// TIA Portal project "CommRS485" (V17)

(* hardware
DEVICE "S7-1200 station_1"  S7-1200 Station
   slot 0: "Rack_0"  S7-1200 Rack  Rack  V1.0
   slot 1: "PLC_1"  CPU 1211C DC/DC/Rly  6ES7 211-1HE40-0XB0  V4.5
   slot 101: "CM 1241 (RS422/485)_1"  6ES7 241-1CH32-0XB0  V2.2
DEVICE "S7-1200 station_2"  S7-1200 Station
   slot 0: "Rack_0"  S7-1200 Rack  Rack  V1.0
   slot 1: "PLC_2"  CPU 1211C DC/DC/Rly  6ES7 211-1HE40-0XB0  V4.5
   slot 101: "CM 1241 (RS422/485)_1"  6ES7 241-1CH32-0XB0  V2.2
DEVICE "S7-1200 station_3"  S7-1200 Station
   slot 0: "Rack_0"  S7-1200 Rack  Rack  V1.0
   slot 1: "PLC_3"  CPU 1214C DC/DC/Rly  6ES7 214-1HG40-0XB0  V4.5
   slot 101: "CM 1241 (RS422/485)_1"  6ES7 241-1CH32-0XB0  V2.2
   slot 102: "CM 1241 (RS422/485)_2"  6ES7 241-1CH32-0XB0  V2.2
*)

// ===== PLC "PLC_1"  CPU 1211C DC/DC/Rly =====

VAR_GLOBAL   // PLC tag table "Default tag table"
   "System_Byte" AT %MB1 : Byte;
   "FirstScan" AT %M1.0 : Bool;
   "DiagStatusUpdate" AT %M1.1 : Bool;
   "AlwaysTRUE" AT %M1.2 : Bool;
   "AlwaysFALSE" AT %M1.3 : Bool;
   "Clock_Byte" AT %MB0 : Byte;
   "Clock_10Hz" AT %M0.0 : Bool;
   "Clock_5Hz" AT %M0.1 : Bool;
   "Clock_2.5Hz" AT %M0.2 : Bool;
   "Clock_2Hz" AT %M0.3 : Bool;
   "Clock_1.25Hz" AT %M0.4 : Bool;
   "Clock_1Hz" AT %M0.5 : Bool;
   "Clock_0.625Hz" AT %M0.6 : Bool;
   "Clock_0.5Hz" AT %M0.7 : Bool;
END_VAR

DATA_BLOCK "MB_LOAD_SLAVE1"   // DB1
{ S7_Optimized_Access := 'FALSE' }
VERSION : 0.1
   VAR
      BAUD : UDInt := 9600;
      PARITY : UInt;
      DONE : Bool;
      ERROR : Bool;
      STATUS : Word;
   END_VAR
BEGIN
END_DATA_BLOCK

DATA_BLOCK "MB_CONFIG_SLAVE"   // DB2
{ S7_Optimized_Access := 'FALSE' }
VERSION : 0.1
   VAR
      MB_ADDR : UInt := 1;
   END_VAR
BEGIN
END_DATA_BLOCK

DATA_BLOCK "DATA_BUFF"   // DB3
{ S7_Optimized_Access := 'FALSE' }
VERSION : 0.1
   VAR
      REGISTRE : Array[0..9] of Bool;
   END_VAR
BEGIN
END_DATA_BLOCK

FUNCTION "Block_1" : Void   // FC1, LAD
{ S7_Optimized_Access := 'TRUE' }
VERSION : 0.1
BEGIN

REGION Network 1
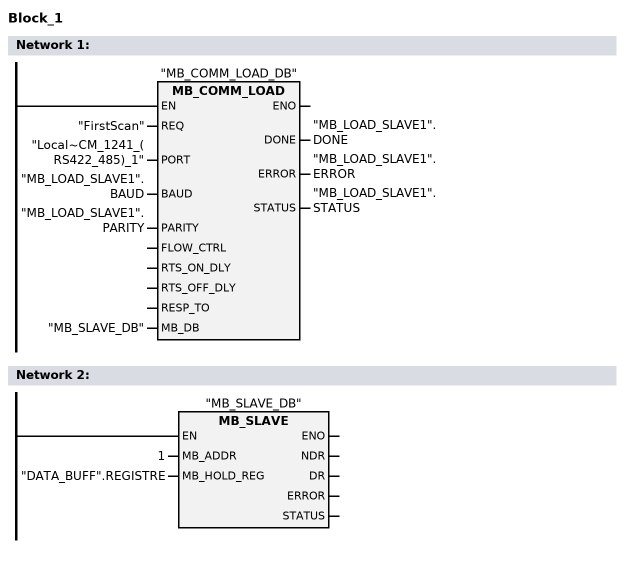
   "MB_COMM_LOAD_DB"(REQ := "FirstScan",   // MB_COMM_LOAD
                     PORT := "Local~CM_1241_(RS422_485)_1",
                     BAUD := "MB_LOAD_SLAVE1".BAUD,
                     PARITY := "MB_LOAD_SLAVE1".PARITY,
                     MB_DB := "MB_SLAVE_DB",
                     DONE => "MB_LOAD_SLAVE1".DONE,
                     ERROR => "MB_LOAD_SLAVE1".ERROR,
                     STATUS => "MB_LOAD_SLAVE1".STATUS);
END_REGION

REGION Network 2
   "MB_SLAVE_DB"(MB_ADDR := 1, MB_HOLD_REG := "DATA_BUFF".REGISTRE);   // MB_SLAVE
END_REGION
END_FUNCTION

ORGANIZATION_BLOCK "Main"   // OB1, LAD, ProgramCycle
TITLE = "Main Program Sweep (Cycle)"
{ S7_Optimized_Access := 'TRUE' }
VERSION : 0.1
   VAR_INPUT
      Initial_Call : Bool;   // Initial call of this OB
      Remanence : Bool;   // =True, if remanent data are available
   END_VAR
BEGIN

REGION Network 1
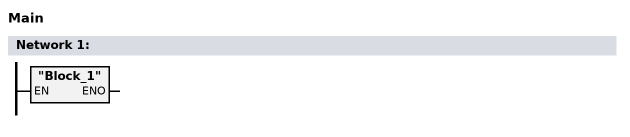
   RUNG wire#powerrail
      "Block_1"()
   END_RUNG
   // the same network as SCL:
   "Block_1"();
END_REGION
END_ORGANIZATION_BLOCK

// ===== PLC "PLC_2"  CPU 1211C DC/DC/Rly =====

VAR_GLOBAL   // PLC tag table "Default tag table"
   "System_Byte" AT %MB1 : Byte;
   "FirstScan" AT %M1.0 : Bool;
   "DiagStatusUpdate" AT %M1.1 : Bool;
   "AlwaysTRUE" AT %M1.2 : Bool;
   "AlwaysFALSE" AT %M1.3 : Bool;
   "Clock_Byte" AT %MB0 : Byte;
   "Clock_10Hz" AT %M0.0 : Bool;
   "Clock_5Hz" AT %M0.1 : Bool;
   "Clock_2.5Hz" AT %M0.2 : Bool;
   "Clock_2Hz" AT %M0.3 : Bool;
   "Clock_1.25Hz" AT %M0.4 : Bool;
   "Clock_1Hz" AT %M0.5 : Bool;
   "Clock_0.625Hz" AT %M0.6 : Bool;
   "Clock_0.5Hz" AT %M0.7 : Bool;
END_VAR

DATA_BLOCK "MB_LOAD_SLAVE1"   // DB1
{ S7_Optimized_Access := 'FALSE' }
VERSION : 0.1
   VAR
      BAUD : UDInt := 9600;
      PARITY : UInt;
      DONE : Bool;
      ERROR : Bool;
      STATUS : Word;
   END_VAR
BEGIN
END_DATA_BLOCK

DATA_BLOCK "MB_CONFIG_SLAVE"   // DB2
{ S7_Optimized_Access := 'FALSE' }
VERSION : 0.1
   VAR
      MB_ADDR : UInt := 2;
   END_VAR
BEGIN
END_DATA_BLOCK

DATA_BLOCK "DATA_BUFF"   // DB3
{ S7_Optimized_Access := 'FALSE' }
VERSION : 0.1
   VAR
      REGISTRE : Array[0..9] of Bool;
   END_VAR
BEGIN
END_DATA_BLOCK

FUNCTION "Block_1" : Void   // FC1, LAD
{ S7_Optimized_Access := 'TRUE' }
VERSION : 0.1
BEGIN

REGION Network 1
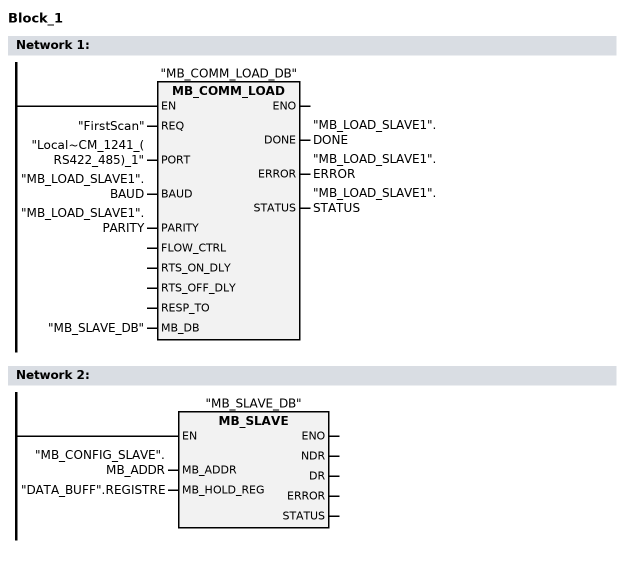
   "MB_COMM_LOAD_DB"(REQ := "FirstScan",   // MB_COMM_LOAD
                     PORT := "Local~CM_1241_(RS422_485)_1",
                     BAUD := "MB_LOAD_SLAVE1".BAUD,
                     PARITY := "MB_LOAD_SLAVE1".PARITY,
                     MB_DB := "MB_SLAVE_DB",
                     DONE => "MB_LOAD_SLAVE1".DONE,
                     ERROR => "MB_LOAD_SLAVE1".ERROR,
                     STATUS => "MB_LOAD_SLAVE1".STATUS);
END_REGION

REGION Network 2
   "MB_SLAVE_DB"(MB_ADDR := "MB_CONFIG_SLAVE".MB_ADDR, MB_HOLD_REG := "DATA_BUFF".REGISTRE);   // MB_SLAVE
END_REGION
END_FUNCTION

ORGANIZATION_BLOCK "Main"   // OB1, LAD, ProgramCycle
TITLE = "Main Program Sweep (Cycle)"
{ S7_Optimized_Access := 'TRUE' }
VERSION : 0.1
   VAR_INPUT
      Initial_Call : Bool;   // Initial call of this OB
      Remanence : Bool;   // =True, if remanent data are available
   END_VAR
BEGIN

REGION Network 1
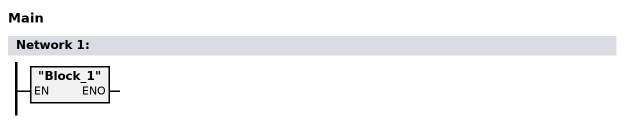
   RUNG wire#powerrail
      "Block_1"()
   END_RUNG
   // the same network as SCL:
   "Block_1"();
END_REGION
END_ORGANIZATION_BLOCK

// ===== PLC "PLC_3"  CPU 1214C DC/DC/Rly =====

VAR_GLOBAL   // PLC tag table "Default tag table"
   "System_Byte" AT %MB1 : Byte;
   "FirstScan" AT %M1.0 : Bool;
   "DiagStatusUpdate" AT %M1.1 : Bool;
   "AlwaysTRUE" AT %M1.2 : Bool;
   "AlwaysFALSE" AT %M1.3 : Bool;
   "Clock_Byte" AT %MB0 : Byte;
   "Clock_10Hz" AT %M0.0 : Bool;
   "Clock_5Hz" AT %M0.1 : Bool;
   "Clock_2.5Hz" AT %M0.2 : Bool;
   "Clock_2Hz" AT %M0.3 : Bool;
   "Clock_1.25Hz" AT %M0.4 : Bool;
   "Clock_1Hz" AT %M0.5 : Bool;
   "Clock_0.625Hz" AT %M0.6 : Bool;
   "Clock_0.5Hz" AT %M0.7 : Bool;
   "Tag_1" AT %M10.0 : Bool;
   "IN0" AT %I0.0 : Bool;
   "IN1" AT %I0.1 : Bool;
   "IN2" AT %I0.2 : Bool;
   "IN3" AT %I0.3 : Bool;
   "IN4" AT %I0.4 : Bool;
   "IN5" AT %I0.5 : Bool;
   "IN6" AT %I0.6 : Bool;
   "IN7" AT %I0.7 : Bool;
   "IN8" AT %I1.0 : Bool;
   "IN9" AT %I1.1 : Bool;
   "IN10" AT %I1.2 : Bool;
   "IN11" AT %I1.3 : Bool;
   "IN12" AT %I1.4 : Bool;
   "IN13" AT %I1.5 : Bool;
   "OUT0" AT %Q0.0 : Bool;
   "OUT1" AT %Q0.1 : Bool;
   "OUT2" AT %Q0.2 : Bool;
   "OUT3" AT %Q0.3 : Bool;
   "OUT4" AT %Q0.4 : Bool;
   "OUT5" AT %Q0.5 : Bool;
   "OUT6" AT %Q0.6 : Bool;
   "OUT7" AT %Q0.7 : Bool;
   "OUT8" AT %Q1.0 : Bool;
   "OUT9" AT %Q1.1 : Bool;
   "ManuE" AT %M20.0 : Bool;
   "ManuS" AT %M20.1 : Bool;
   "CmdE" AT %M20.2 : Bool;
   "CmdS" AT %M20.3 : Bool;
   "AutoE" AT %M20.4 : Bool;
   "AutoS" AT %M20.5 : Bool;
   "RBE" AT %M20.6 : Bool;
   "RBS" AT %M20.7 : Bool;
   "C1E" AT %M21.0 : Bool;
   "C2E" AT %M21.1 : Bool;
   "C3E" AT %M21.2 : Bool;
   "C1S" AT %M21.3 : Bool;
   "C2S" AT %M21.4 : Bool;
   "B1" AT %M21.5 : Bool;
   "B2" AT %M21.6 : Bool;
   "B3" AT %M21.7 : Bool;
   "B4" AT %M22.0 : Bool;
   "BPBE" AT %M22.1 : Bool;
   "BPBS" AT %M22.2 : Bool;
   "CBE" AT %M22.3 : Bool;
   "CBS" AT %M22.4 : Bool;
   "URG" AT %M22.5 : Bool;
   "MRBE" AT %M30.0 : Bool;
   "MRBS" AT %M30.1 : Bool;
   "DRBE" AT %M30.2 : Bool;
   "DRBS" AT %M30.3 : Bool;
   "FVE" AT %M30.4 : Bool;
   "FVS" AT %M30.5 : Bool;
   "BME" AT %M30.6 : Bool;
   "BMS" AT %M30.7 : Bool;
   "X0" AT %M40.0 : Bool;
   "X1" AT %M40.1 : Bool;
   "X2" AT %M40.2 : Bool;
   "X3" AT %M40.3 : Bool;
   "X10" AT %M40.4 : Bool;
   "X11" AT %M40.5 : Bool;
   "X12" AT %M40.6 : Bool;
   "X13" AT %M40.7 : Bool;
   "X14" AT %M41.0 : Bool;
   "X15" AT %M41.1 : Bool;
   "X16" AT %M41.2 : Bool;
   "X17" AT %M41.3 : Bool;
   "X20" AT %M41.4 : Bool;
   "X21" AT %M41.5 : Bool;
   "X30" AT %M41.6 : Bool;
   "X31" AT %M41.7 : Bool;
   "X32" AT %M42.0 : Bool;
   "X33" AT %M42.1 : Bool;
   "X40" AT %M42.2 : Bool;
   "X41" AT %M42.3 : Bool;
   "X42" AT %M42.4 : Bool;
   "X43" AT %M42.5 : Bool;
   "X44" AT %M42.6 : Bool;
   "X45" AT %M42.7 : Bool;
   "X50" AT %M43.0 : Bool;
   "X51" AT %M43.1 : Bool;
   "X60" AT %M43.2 : Bool;
   "X61" AT %M43.3 : Bool;
   "X62" AT %M43.4 : Bool;
   "X63" AT %M43.5 : Bool;
   "X70" AT %M43.6 : Bool;
   "X71" AT %M43.7 : Bool;
   "X72" AT %M44.0 : Bool;
   "X73" AT %M44.1 : Bool;
   "X80" AT %M44.2 : Bool;
   "X81" AT %M44.3 : Bool;
   "C1" AT %M31.0 : Bool;
   "C2" AT %M31.1 : Bool;
   "F10" AT %M44.4 : Bool;
   "F20" AT %M44.5 : Bool;
   "F30" AT %M44.6 : Bool;
   "F0" AT %M44.7 : Bool;
   "F50" AT %M45.0 : Bool;
   "F40" AT %M45.1 : Bool;
   "F60" AT %M45.2 : Bool;
   "F70" AT %M45.3 : Bool;
   "C1E_Memo" AT %M70.0 : Bool;
   "C2E_Memo" AT %M70.1 : Bool;
   "C3E_Memo" AT %M70.2 : Bool;
   "C1S_Memo" AT %M70.3 : Bool;
   "C2S_Memo" AT %M70.4 : Bool;
   "IN14" AT %I1.6 : Bool;
   "X18" AT %M45.5 : Bool;
   "X4" AT %M45.6 : Bool;
   "X64" AT %M45.7 : Bool;
   "X65" AT %M46.0 : Bool;
   "X46" AT %M46.1 : Bool;
   "X47" AT %M46.2 : Bool;
   "X48" AT %M46.3 : Bool;
   "X49" AT %M46.4 : Bool;
   "C1S_Memo2" AT %M46.5 : Bool;
   "C2S_Memo2" AT %M46.6 : Bool;
   "C1E_Memo2" AT %M46.7 : Bool;
   "C2E_Memo2" AT %M47.0 : Bool;
   "C3E_Memo2" AT %M47.1 : Bool;
   "FRE" AT %M47.2 : Bool;
   "FRS" AT %M47.3 : Bool;
   "X66" AT %M47.4 : Bool;
   "X34" AT %M47.5 : Bool;
   "X74" AT %M47.6 : Bool;
   "X75" AT %M47.7 : Bool;
   "T1" AT %M48.0 : Bool;
   "T2" AT %M48.1 : Bool;
   "T3" AT %M48.2 : Bool;
   "T4" AT %M48.3 : Bool;
   "T5" AT %M48.4 : Bool;
   "T6" AT %M48.5 : Bool;
   "T7" AT %M48.6 : Bool;
   "T8" AT %M48.7 : Bool;
   "T9" AT %M49.0 : Bool;
   "T10" AT %M49.1 : Bool;
   "X90" AT %M49.2 : Bool;
   "X91" AT %M49.3 : Bool;
   "index1E" AT %MW49 : Int;
   "index2E" AT %MW50 : Int;
   "Index1S" AT %MW51 : Int;
   "index2S" AT %MW52 : Int;
   "memoCmd" AT %M54.0 : Bool;
   "memoX10" AT %M54.1 : Bool;
   "TestCmd" AT %M54.2 : Bool;
   "memoTestCmd" AT %M54.3 : Bool;
   "BFE" AT %M54.4 : Bool;
   "BFS" AT %M54.5 : Bool;
   "TestX40" AT %M54.6 : Bool;
END_VAR

DATA_BLOCK "MBLOAD_MatserReadSlave1"   // DB1
{ S7_Optimized_Access := 'FALSE' }
VERSION : 0.1
   VAR
      Baud : UDInt := 9600;
      PARITY : UInt;
      DONE : Bool;
      ERROR : Bool;
      STATUS : Word;
   END_VAR
BEGIN
END_DATA_BLOCK

DATA_BLOCK "MBCONFIG_MasterReadSlave1"   // DB2
{ S7_Optimized_Access := 'FALSE' }
VERSION : 0.1
   VAR
      REQ : Bool;
      AGAIN : Bool;
      MB_ADDR : UInt := 1;
      MODE : USInt;
      DATA_ADDR : UDInt := 10001;
      DATA_LEN : UInt := 10;
      DONE : Bool;
      ERROR : Bool;
      BUSY : Bool;
      Register_Input : Array[0..9] of Bool;
      STATUS : Word;
   END_VAR
BEGIN
END_DATA_BLOCK

DATA_BLOCK "DATA_BUFF_InputSlave1"   // DB3
{ S7_Optimized_Access := 'FALSE' }
VERSION : 0.1
   VAR
      REGISTERS : Array[0..9] of Bool;
   END_VAR
BEGIN
END_DATA_BLOCK

DATA_BLOCK "MBLOAD_MatserReadSlave2"   // DB7
{ S7_Optimized_Access := 'FALSE' }
VERSION : 0.1
   VAR
      Baud : UDInt := 9600;
      PARITY : UInt;
      DONE : Bool;
      ERROR : Bool;
      STATUS : Word;
   END_VAR
BEGIN
END_DATA_BLOCK

DATA_BLOCK "MBCONFIG_MasterReadSlave2"   // DB8
{ S7_Optimized_Access := 'FALSE' }
VERSION : 0.1
   VAR
      REQ : Bool;
      AGAIN : Bool;
      MB_ADDR : UInt := 2;
      MODE : USInt;
      DATA_ADDR : UDInt := 10001;
      DATA_LEN : UInt := 10;
      DONE : Bool;
      ERROR : Bool;
      BUSY : Bool;
      Register_Input : Array[0..9] of Bool;
      STATUS : Word;
   END_VAR
BEGIN
END_DATA_BLOCK

DATA_BLOCK "Data_BUFF_InputSlave2"   // DB9
{ S7_Optimized_Access := 'FALSE' }
VERSION : 0.1
   VAR
      REGISTERS : Array[0..9] of Bool;
   END_VAR
BEGIN
END_DATA_BLOCK

DATA_BLOCK "Data_Buff_OutputSlave1"   // DB10
{ S7_Optimized_Access := 'FALSE' }
VERSION : 0.1
   VAR
      Register : Array[0..9] of Bool;
   END_VAR
BEGIN
END_DATA_BLOCK

DATA_BLOCK "Data_Buff_OutputSlave2"   // DB11
{ S7_Optimized_Access := 'FALSE' }
VERSION : 0.1
   VAR
      Register : Array[0..9] of Bool;
   END_VAR
BEGIN
END_DATA_BLOCK

DATA_BLOCK "MBCONFIG_MasterWriteSlave1"   // DB12
{ S7_Optimized_Access := 'FALSE' }
VERSION : 0.1
   VAR
      REQ : Bool;
      AGAIN : Bool;
      MB_ADDR : UInt := 1;
      MODE : USInt := 1;
      DATA_ADDR : UDInt := 1;
      DATA_LEN : UInt := 10;
      DONE : Bool;
      ERROR : Bool;
      BUSY : Bool;
      Register_Input : Array[0..9] of Bool;
      STATUS : Word;
   END_VAR
BEGIN
END_DATA_BLOCK

DATA_BLOCK "MBCONFIG_MasterWriteSlave2"   // DB13
{ S7_Optimized_Access := 'FALSE' }
VERSION : 0.1
   VAR
      REQ : Bool;
      AGAIN : Bool;
      MB_ADDR : UInt := 2;
      MODE : USInt := 1;
      DATA_ADDR : UDInt := 1;
      DATA_LEN : UInt := 10;
      DONE : Bool;
      ERROR : Bool;
      BUSY : Bool;
      Register_Input : Array[0..9] of Bool;
      STATUS : Word;
   END_VAR
BEGIN
END_DATA_BLOCK

DATA_BLOCK "MBLOAD_MatserWriteSlave1"   // DB14
{ S7_Optimized_Access := 'FALSE' }
VERSION : 0.1
   VAR
      Baud : UDInt := 9600;
      PARITY : UInt := 0;
      DONE : Bool;
      ERROR : Bool;
      STATUS : Word;
   END_VAR
BEGIN
END_DATA_BLOCK

DATA_BLOCK "MBLOAD_MatserWriteSlave2"   // DB15
{ S7_Optimized_Access := 'FALSE' }
VERSION : 0.1
   VAR
      Baud : UDInt := 9600;
      PARITY : UInt := 1;
      DONE : Bool;
      ERROR : Bool;
      STATUS : Word;
   END_VAR
BEGIN
END_DATA_BLOCK

DATA_BLOCK "CMD"   // DB28
{ S7_Optimized_Access := 'FALSE' }
VERSION : 0.1
   VAR
      CMDE : Array[0..4] of Bool;
      CMDFinal_E : Bool;
      CMDS : Array[0..4] of Bool;
      CMDFinal_S : Bool;
   END_VAR
BEGIN
END_DATA_BLOCK

// folder: System blocks/Program resources

DATA_BLOCK "IEC_Timer_0_DB"   // DB16
{ S7_Optimized_Access := 'TRUE' }
AUTHOR : Simatic
FAMILY : IEC
NAME : IEC_TMR
VERSION : 1.0
// stored: InstanceOfName IEC_TIMER
"IEC_TIMER"
BEGIN
END_DATA_BLOCK

DATA_BLOCK "IEC_Timer_0_DB_1"   // DB19
{ S7_Optimized_Access := 'TRUE' }
AUTHOR : Simatic
FAMILY : IEC
NAME : IEC_TMR
VERSION : 1.0
// stored: InstanceOfName IEC_TIMER
"IEC_TIMER"
BEGIN
END_DATA_BLOCK

DATA_BLOCK "IEC_Timer_0_DB_2"   // DB21
{ S7_Optimized_Access := 'TRUE' }
AUTHOR : Simatic
FAMILY : IEC
NAME : IEC_TMR
VERSION : 1.0
// stored: InstanceOfName IEC_TIMER
"IEC_TIMER"
BEGIN
END_DATA_BLOCK

DATA_BLOCK "IEC_Timer_0_DB_3"   // DB24
{ S7_Optimized_Access := 'TRUE' }
AUTHOR : Simatic
FAMILY : IEC
NAME : IEC_TMR
VERSION : 1.0
// stored: InstanceOfName IEC_TIMER
"IEC_TIMER"
BEGIN
END_DATA_BLOCK

DATA_BLOCK "IEC_Timer_0_DB_4"   // DB25
{ S7_Optimized_Access := 'TRUE' }
AUTHOR : Simatic
FAMILY : IEC
NAME : IEC_TMR
VERSION : 1.0
// stored: InstanceOfName IEC_TIMER
"IEC_TIMER"
BEGIN
END_DATA_BLOCK

DATA_BLOCK "IEC_Timer_0_DB_5"   // DB26
{ S7_Optimized_Access := 'TRUE' }
AUTHOR : Simatic
FAMILY : IEC
NAME : IEC_TMR
VERSION : 1.0
// stored: InstanceOfName IEC_TIMER
"IEC_TIMER"
BEGIN
END_DATA_BLOCK

DATA_BLOCK "IEC_Timer_0_DB_6"   // DB27
{ S7_Optimized_Access := 'TRUE' }
AUTHOR : Simatic
FAMILY : IEC
NAME : IEC_TMR
VERSION : 1.0
// stored: InstanceOfName IEC_TIMER
"IEC_TIMER"
BEGIN
END_DATA_BLOCK

DATA_BLOCK "IEC_Timer_0_DB_8"   // DB29
{ S7_Optimized_Access := 'TRUE' }
AUTHOR : Simatic
FAMILY : IEC
NAME : IEC_TMR
VERSION : 1.0
// stored: InstanceOfName IEC_TIMER
"IEC_TIMER"
BEGIN
END_DATA_BLOCK

DATA_BLOCK "IEC_Timer_0_DB_9"   // DB30
{ S7_Optimized_Access := 'TRUE' }
AUTHOR : Simatic
FAMILY : IEC
NAME : IEC_TMR
VERSION : 1.0
// stored: InstanceOfName IEC_TIMER
"IEC_TIMER"
BEGIN
END_DATA_BLOCK

DATA_BLOCK "IEC_Timer_0_DB_11"   // DB32
{ S7_Optimized_Access := 'TRUE' }
AUTHOR : Simatic
FAMILY : IEC
NAME : IEC_TMR
VERSION : 1.0
// stored: InstanceOfName IEC_TIMER
"IEC_TIMER"
BEGIN
END_DATA_BLOCK

DATA_BLOCK "IEC_Timer_0_DB_13"   // DB34
{ S7_Optimized_Access := 'TRUE' }
AUTHOR : Simatic
FAMILY : IEC
NAME : IEC_TMR
VERSION : 1.0
// stored: InstanceOfName IEC_TIMER
"IEC_TIMER"
BEGIN
END_DATA_BLOCK

// folder: (top level)

FUNCTION "REQ_Master_To_Slave1" : Void   // FC1, LAD
{ S7_Optimized_Access := 'TRUE' }
VERSION : 0.1
BEGIN

REGION Network 1: Lecture des entrées
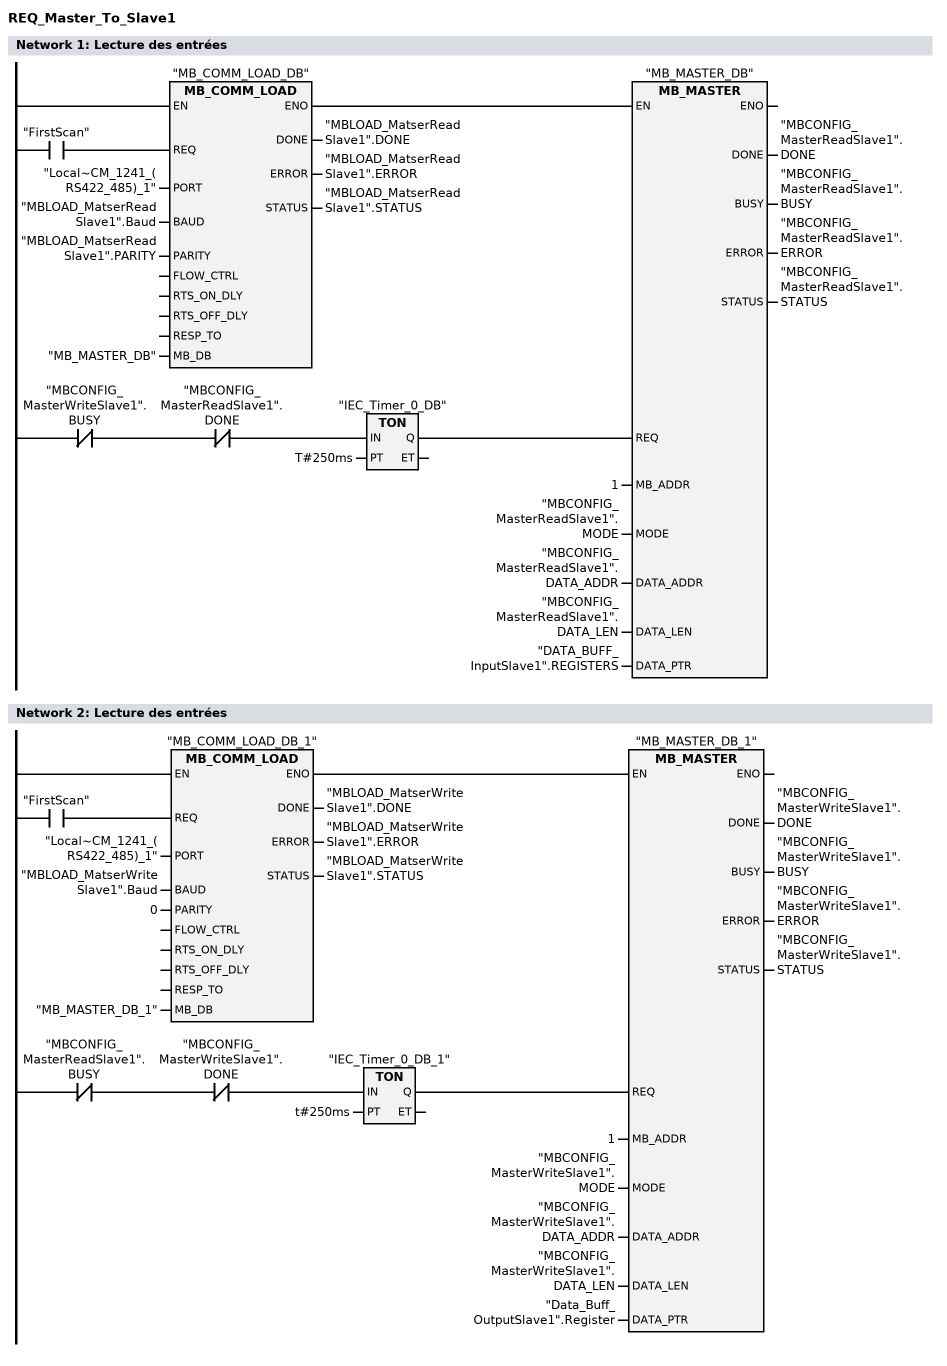
   // ENO of a box is taken as its EN; it also drops when the box reports an error
   "MB_COMM_LOAD_DB"(REQ := "FirstScan",   // MB_COMM_LOAD
                     PORT := "Local~CM_1241_(RS422_485)_1",
                     BAUD := "MBLOAD_MatserReadSlave1".Baud,
                     PARITY := "MBLOAD_MatserReadSlave1".PARITY,
                     MB_DB := "MB_MASTER_DB",
                     DONE => "MBLOAD_MatserReadSlave1".DONE,
                     ERROR => "MBLOAD_MatserReadSlave1".ERROR,
                     STATUS => "MBLOAD_MatserReadSlave1".STATUS);
   "IEC_Timer_0_DB".TON(IN := NOT "MBCONFIG_MasterWriteSlave1".BUSY AND NOT "MBCONFIG_MasterReadSlave1".DONE,
                        PT := T#250ms);
   "MB_MASTER_DB"(REQ := "IEC_Timer_0_DB".Q,   // MB_MASTER
                  MB_ADDR := 1,
                  MODE := "MBCONFIG_MasterReadSlave1".MODE,
                  DATA_ADDR := "MBCONFIG_MasterReadSlave1".DATA_ADDR,
                  DATA_LEN := "MBCONFIG_MasterReadSlave1".DATA_LEN,
                  DATA_PTR := "DATA_BUFF_InputSlave1".REGISTERS,
                  DONE => "MBCONFIG_MasterReadSlave1".DONE,
                  BUSY => "MBCONFIG_MasterReadSlave1".BUSY,
                  ERROR => "MBCONFIG_MasterReadSlave1".ERROR,
                  STATUS => "MBCONFIG_MasterReadSlave1".STATUS);
END_REGION

REGION Network 2: Lecture des entrées
   // ENO of a box is taken as its EN; it also drops when the box reports an error
   "MB_COMM_LOAD_DB_1"(REQ := "FirstScan",   // MB_COMM_LOAD
                       PORT := "Local~CM_1241_(RS422_485)_1",
                       BAUD := "MBLOAD_MatserWriteSlave1".Baud,
                       PARITY := 0,
                       MB_DB := "MB_MASTER_DB_1",
                       DONE => "MBLOAD_MatserWriteSlave1".DONE,
                       ERROR => "MBLOAD_MatserWriteSlave1".ERROR,
                       STATUS => "MBLOAD_MatserWriteSlave1".STATUS);
   "IEC_Timer_0_DB_1".TON(IN := NOT "MBCONFIG_MasterReadSlave1".BUSY AND NOT "MBCONFIG_MasterWriteSlave1".DONE,
                          PT := t#250ms);
   "MB_MASTER_DB_1"(REQ := "IEC_Timer_0_DB_1".Q,   // MB_MASTER
                    MB_ADDR := 1,
                    MODE := "MBCONFIG_MasterWriteSlave1".MODE,
                    DATA_ADDR := "MBCONFIG_MasterWriteSlave1".DATA_ADDR,
                    DATA_LEN := "MBCONFIG_MasterWriteSlave1".DATA_LEN,
                    DATA_PTR := "Data_Buff_OutputSlave1".Register,
                    DONE => "MBCONFIG_MasterWriteSlave1".DONE,
                    BUSY => "MBCONFIG_MasterWriteSlave1".BUSY,
                    ERROR => "MBCONFIG_MasterWriteSlave1".ERROR,
                    STATUS => "MBCONFIG_MasterWriteSlave1".STATUS);
END_REGION
END_FUNCTION

FUNCTION "REQ_Master_To_Slave2" : Void   // FC2, LAD
{ S7_Optimized_Access := 'TRUE' }
VERSION : 0.1
BEGIN

REGION Network 1: LECTURE ENTREES
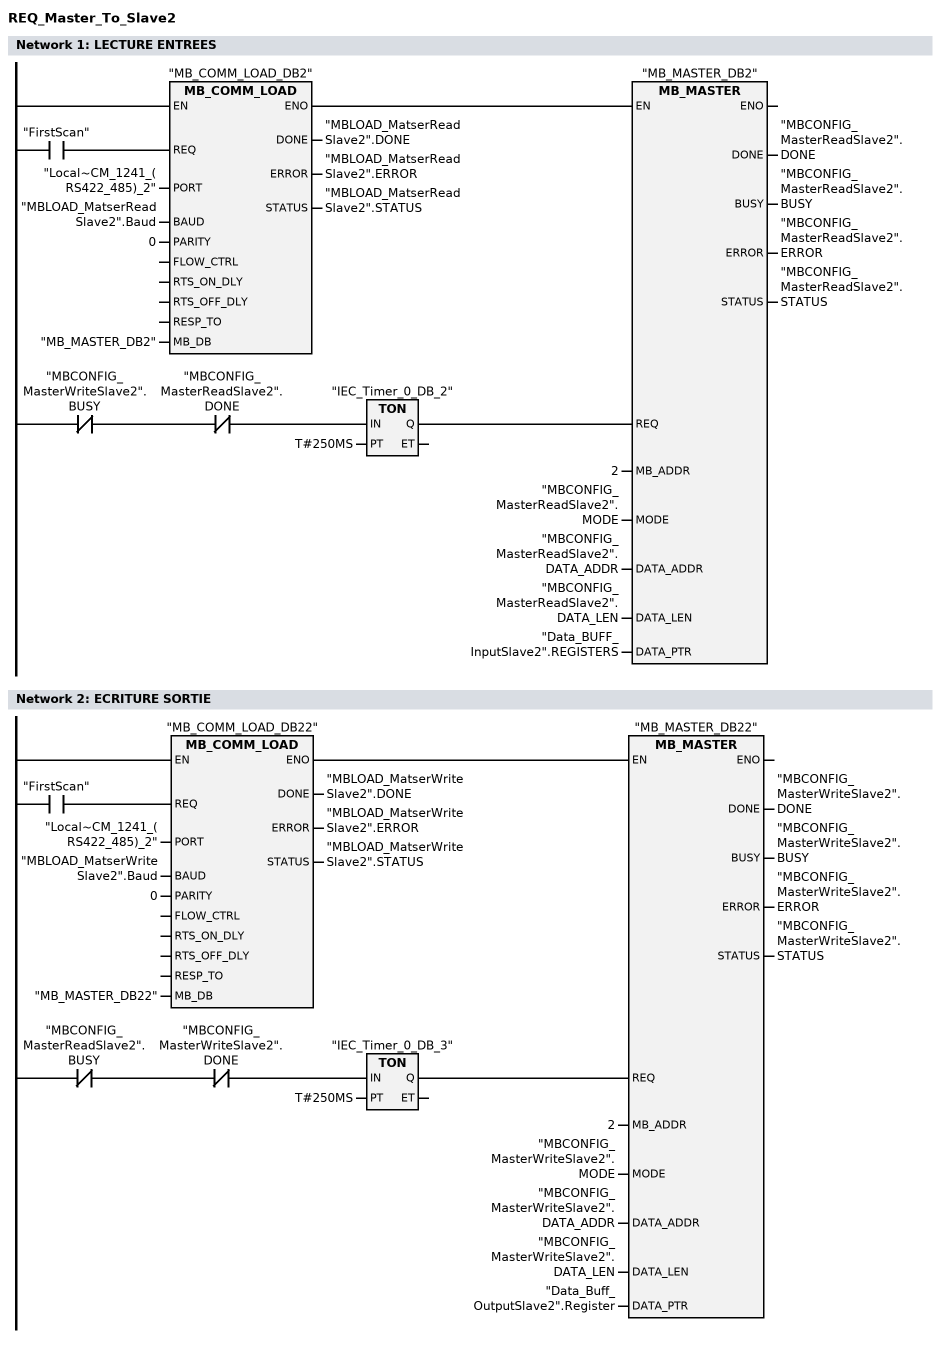
   // ENO of a box is taken as its EN; it also drops when the box reports an error
   "MB_COMM_LOAD_DB2"(REQ := "FirstScan",   // MB_COMM_LOAD
                      PORT := "Local~CM_1241_(RS422_485)_2",
                      BAUD := "MBLOAD_MatserReadSlave2".Baud,
                      PARITY := 0,
                      MB_DB := "MB_MASTER_DB2",
                      DONE => "MBLOAD_MatserReadSlave2".DONE,
                      ERROR => "MBLOAD_MatserReadSlave2".ERROR,
                      STATUS => "MBLOAD_MatserReadSlave2".STATUS);
   "IEC_Timer_0_DB_2".TON(IN := NOT "MBCONFIG_MasterWriteSlave2".BUSY AND NOT "MBCONFIG_MasterReadSlave2".DONE,
                          PT := T#250MS);
   "MB_MASTER_DB2"(REQ := "IEC_Timer_0_DB_2".Q,   // MB_MASTER
                   MB_ADDR := 2,
                   MODE := "MBCONFIG_MasterReadSlave2".MODE,
                   DATA_ADDR := "MBCONFIG_MasterReadSlave2".DATA_ADDR,
                   DATA_LEN := "MBCONFIG_MasterReadSlave2".DATA_LEN,
                   DATA_PTR := "Data_BUFF_InputSlave2".REGISTERS,
                   DONE => "MBCONFIG_MasterReadSlave2".DONE,
                   BUSY => "MBCONFIG_MasterReadSlave2".BUSY,
                   ERROR => "MBCONFIG_MasterReadSlave2".ERROR,
                   STATUS => "MBCONFIG_MasterReadSlave2".STATUS);
END_REGION

REGION Network 2: ECRITURE SORTIE
   // ENO of a box is taken as its EN; it also drops when the box reports an error
   "MB_COMM_LOAD_DB22"(REQ := "FirstScan",   // MB_COMM_LOAD
                       PORT := "Local~CM_1241_(RS422_485)_2",
                       BAUD := "MBLOAD_MatserWriteSlave2".Baud,
                       PARITY := 0,
                       MB_DB := "MB_MASTER_DB22",
                       DONE => "MBLOAD_MatserWriteSlave2".DONE,
                       ERROR => "MBLOAD_MatserWriteSlave2".ERROR,
                       STATUS => "MBLOAD_MatserWriteSlave2".STATUS);
   "IEC_Timer_0_DB_3".TON(IN := NOT "MBCONFIG_MasterReadSlave2".BUSY AND NOT "MBCONFIG_MasterWriteSlave2".DONE,
                          PT := T#250MS);
   "MB_MASTER_DB22"(REQ := "IEC_Timer_0_DB_3".Q,   // MB_MASTER
                    MB_ADDR := 2,
                    MODE := "MBCONFIG_MasterWriteSlave2".MODE,
                    DATA_ADDR := "MBCONFIG_MasterWriteSlave2".DATA_ADDR,
                    DATA_LEN := "MBCONFIG_MasterWriteSlave2".DATA_LEN,
                    DATA_PTR := "Data_Buff_OutputSlave2".Register,
                    DONE => "MBCONFIG_MasterWriteSlave2".DONE,
                    BUSY => "MBCONFIG_MasterWriteSlave2".BUSY,
                    ERROR => "MBCONFIG_MasterWriteSlave2".ERROR,
                    STATUS => "MBCONFIG_MasterWriteSlave2".STATUS);
END_REGION
END_FUNCTION

FUNCTION "ConduiteE" : Void   // FC3, LAD
{ S7_Optimized_Access := 'TRUE' }
VERSION : 0.1
BEGIN

REGION Network 1
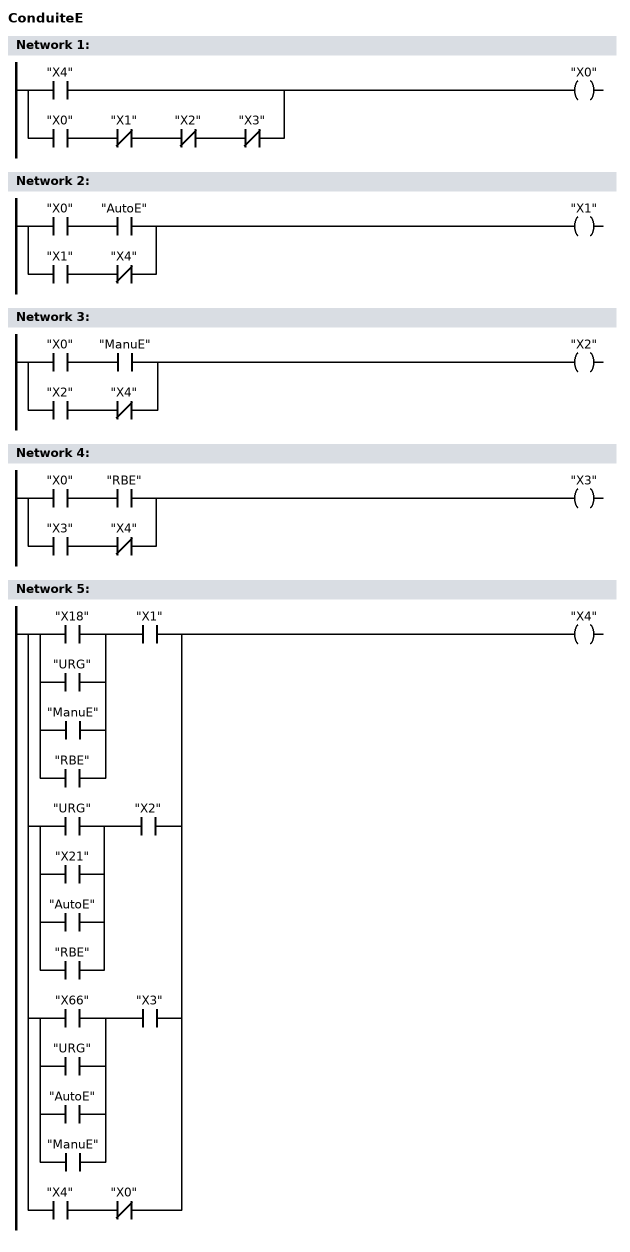
   RUNG wire#powerrail
      Contact( "X4" )
      wire#w1
      Coil( "X0" )
   END_RUNG
   RUNG wire#powerrail
      Contact( "X0" )
      I_Contact( "X1" )
      I_Contact( "X2" )
      I_Contact( "X3" )
   END_RUNG wire#w1
   // the same network as SCL:
   "X0" := "X4" OR ("X0" AND NOT "X1" AND NOT "X2" AND NOT "X3");
END_REGION

REGION Network 2
   RUNG wire#powerrail
      Contact( "X0" )
      Contact( "AutoE" )
      wire#w1
      Coil( "X1" )
   END_RUNG
   RUNG wire#powerrail
      Contact( "X1" )
      I_Contact( "X4" )
   END_RUNG wire#w1
   // the same network as SCL:
   "X1" := ("X0" AND "AutoE") OR ("X1" AND NOT "X4");
END_REGION

REGION Network 3
   RUNG wire#powerrail
      Contact( "X0" )
      Contact( "ManuE" )
      wire#w1
      Coil( "X2" )
   END_RUNG
   RUNG wire#powerrail
      Contact( "X2" )
      I_Contact( "X4" )
   END_RUNG wire#w1
   // the same network as SCL:
   "X2" := ("X0" AND "ManuE") OR ("X2" AND NOT "X4");
END_REGION

REGION Network 4
   RUNG wire#powerrail
      Contact( "X0" )
      Contact( "RBE" )
      wire#w1
      Coil( "X3" )
   END_RUNG
   RUNG wire#powerrail
      Contact( "X3" )
      I_Contact( "X4" )
   END_RUNG wire#w1
   // the same network as SCL:
   "X3" := ("X0" AND "RBE") OR ("X3" AND NOT "X4");
END_REGION

REGION Network 5
   RUNG wire#powerrail
      Contact( "X18" )
      wire#w1
      Contact( "X1" )
      wire#w2
      Coil( "X4" )
   END_RUNG
   RUNG wire#powerrail
      Contact( "URG" )
   END_RUNG wire#w1
   RUNG wire#powerrail
      Contact( "ManuE" )
   END_RUNG wire#w1
   RUNG wire#powerrail
      Contact( "RBE" )
   END_RUNG wire#w1
   RUNG wire#powerrail
      Contact( "URG" )
      wire#w3
      Contact( "X2" )
   END_RUNG wire#w2
   RUNG wire#powerrail
      Contact( "X21" )
   END_RUNG wire#w3
   RUNG wire#powerrail
      Contact( "AutoE" )
   END_RUNG wire#w3
   RUNG wire#powerrail
      Contact( "RBE" )
   END_RUNG wire#w3
   RUNG wire#powerrail
      Contact( "X66" )
      wire#w4
      Contact( "X3" )
   END_RUNG wire#w2
   RUNG wire#powerrail
      Contact( "URG" )
   END_RUNG wire#w4
   RUNG wire#powerrail
      Contact( "AutoE" )
   END_RUNG wire#w4
   RUNG wire#powerrail
      Contact( "ManuE" )
   END_RUNG wire#w4
   RUNG wire#powerrail
      Contact( "X4" )
      I_Contact( "X0" )
   END_RUNG wire#w2
   // the same network as SCL:
   "X4" := (("X18" OR "URG" OR "ManuE" OR "RBE") AND "X1") OR (("URG" OR "X21" OR "AutoE" OR "RBE") AND "X2") OR (("X66" OR "URG" OR "AutoE" OR "ManuE") AND "X3") OR ("X4" AND NOT "X0");
END_REGION
END_FUNCTION

FUNCTION "ConduiteS" : Void   // FC4, LAD
{ S7_Optimized_Access := 'TRUE' }
VERSION : 0.1
BEGIN

REGION Network 1
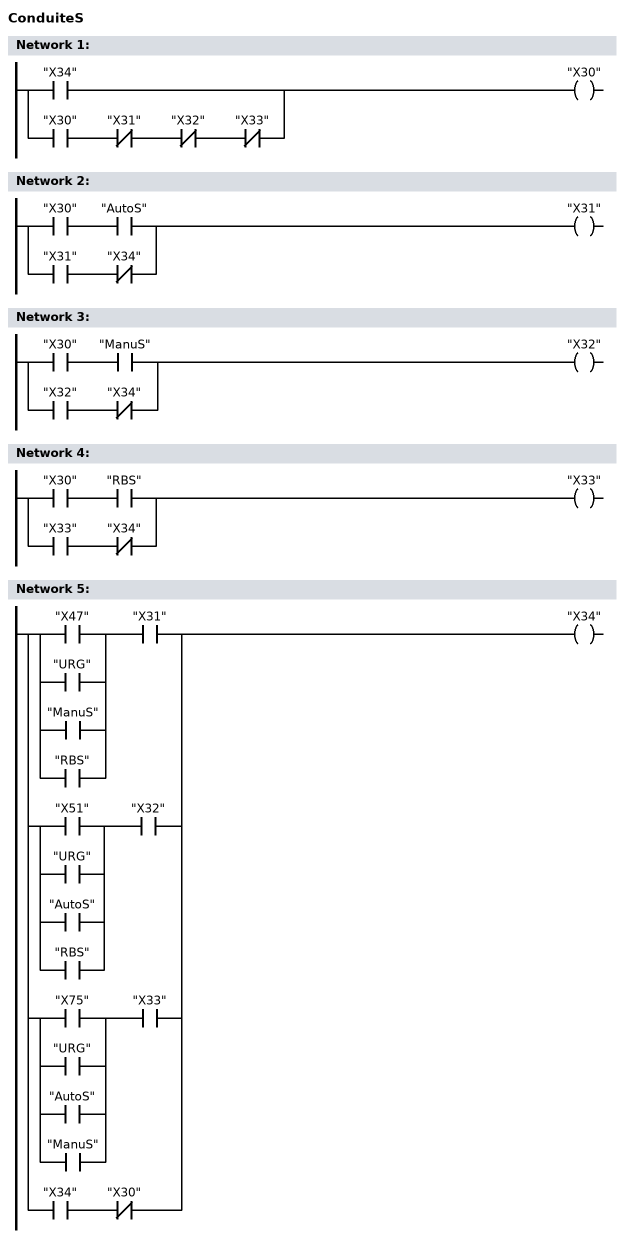
   RUNG wire#powerrail
      Contact( "X34" )
      wire#w1
      Coil( "X30" )
   END_RUNG
   RUNG wire#powerrail
      Contact( "X30" )
      I_Contact( "X31" )
      I_Contact( "X32" )
      I_Contact( "X33" )
   END_RUNG wire#w1
   // the same network as SCL:
   "X30" := "X34" OR ("X30" AND NOT "X31" AND NOT "X32" AND NOT "X33");
END_REGION

REGION Network 2
   RUNG wire#powerrail
      Contact( "X30" )
      Contact( "AutoS" )
      wire#w1
      Coil( "X31" )
   END_RUNG
   RUNG wire#powerrail
      Contact( "X31" )
      I_Contact( "X34" )
   END_RUNG wire#w1
   // the same network as SCL:
   "X31" := ("X30" AND "AutoS") OR ("X31" AND NOT "X34");
END_REGION

REGION Network 3
   RUNG wire#powerrail
      Contact( "X30" )
      Contact( "ManuS" )
      wire#w1
      Coil( "X32" )
   END_RUNG
   RUNG wire#powerrail
      Contact( "X32" )
      I_Contact( "X34" )
   END_RUNG wire#w1
   // the same network as SCL:
   "X32" := ("X30" AND "ManuS") OR ("X32" AND NOT "X34");
END_REGION

REGION Network 4
   RUNG wire#powerrail
      Contact( "X30" )
      Contact( "RBS" )
      wire#w1
      Coil( "X33" )
   END_RUNG
   RUNG wire#powerrail
      Contact( "X33" )
      I_Contact( "X34" )
   END_RUNG wire#w1
   // the same network as SCL:
   "X33" := ("X30" AND "RBS") OR ("X33" AND NOT "X34");
END_REGION

REGION Network 5
   RUNG wire#powerrail
      Contact( "X47" )
      wire#w1
      Contact( "X31" )
      wire#w2
      Coil( "X34" )
   END_RUNG
   RUNG wire#powerrail
      Contact( "URG" )
   END_RUNG wire#w1
   RUNG wire#powerrail
      Contact( "ManuS" )
   END_RUNG wire#w1
   RUNG wire#powerrail
      Contact( "RBS" )
   END_RUNG wire#w1
   RUNG wire#powerrail
      Contact( "X51" )
      wire#w3
      Contact( "X32" )
   END_RUNG wire#w2
   RUNG wire#powerrail
      Contact( "URG" )
   END_RUNG wire#w3
   RUNG wire#powerrail
      Contact( "AutoS" )
   END_RUNG wire#w3
   RUNG wire#powerrail
      Contact( "RBS" )
   END_RUNG wire#w3
   RUNG wire#powerrail
      Contact( "X75" )
      wire#w4
      Contact( "X33" )
   END_RUNG wire#w2
   RUNG wire#powerrail
      Contact( "URG" )
   END_RUNG wire#w4
   RUNG wire#powerrail
      Contact( "AutoS" )
   END_RUNG wire#w4
   RUNG wire#powerrail
      Contact( "ManuS" )
   END_RUNG wire#w4
   RUNG wire#powerrail
      Contact( "X34" )
      I_Contact( "X30" )
   END_RUNG wire#w2
   // the same network as SCL:
   "X34" := (("X47" OR "URG" OR "ManuS" OR "RBS") AND "X31") OR (("X51" OR "URG" OR "AutoS" OR "RBS") AND "X32") OR (("X75" OR "URG" OR "AutoS" OR "ManuS") AND "X33") OR ("X34" AND NOT "X30");
END_REGION
END_FUNCTION

FUNCTION "Manu_E" : Void   // FC5, LAD
{ S7_Optimized_Access := 'TRUE' }
VERSION : 0.1
BEGIN

REGION Network 1
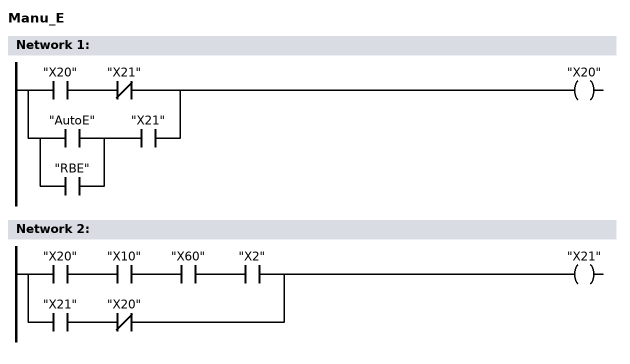
   RUNG wire#powerrail
      Contact( "X20" )
      I_Contact( "X21" )
      wire#w1
      Coil( "X20" )
   END_RUNG
   RUNG wire#powerrail
      Contact( "AutoE" )
      wire#w2
      Contact( "X21" )
   END_RUNG wire#w1
   RUNG wire#powerrail
      Contact( "RBE" )
   END_RUNG wire#w2
   // the same network as SCL:
   "X20" := ("X20" AND NOT "X21") OR (("AutoE" OR "RBE") AND "X21");
END_REGION

REGION Network 2
   RUNG wire#powerrail
      Contact( "X20" )
      Contact( "X10" )
      Contact( "X60" )
      Contact( "X2" )
      wire#w1
      Coil( "X21" )
   END_RUNG
   RUNG wire#powerrail
      Contact( "X21" )
      I_Contact( "X20" )
   END_RUNG wire#w1
   // the same network as SCL:
   "X21" := ("X20" AND "X10" AND "X60" AND "X2") OR ("X21" AND NOT "X20");
END_REGION
END_FUNCTION

FUNCTION "Manu_S" : Void   // FC6, LAD
{ S7_Optimized_Access := 'TRUE' }
VERSION : 0.1
BEGIN

REGION Network 1
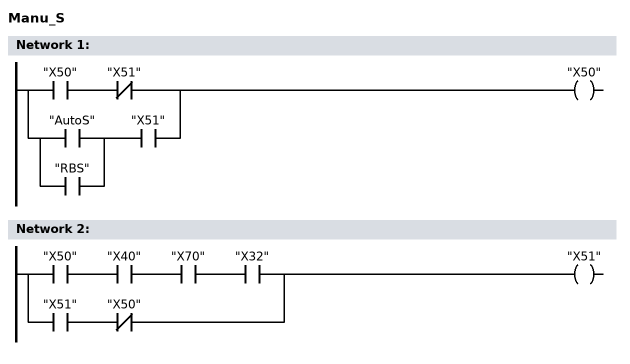
   RUNG wire#powerrail
      Contact( "X50" )
      I_Contact( "X51" )
      wire#w1
      Coil( "X50" )
   END_RUNG
   RUNG wire#powerrail
      Contact( "AutoS" )
      wire#w2
      Contact( "X51" )
   END_RUNG wire#w1
   RUNG wire#powerrail
      Contact( "RBS" )
   END_RUNG wire#w2
   // the same network as SCL:
   "X50" := ("X50" AND NOT "X51") OR (("AutoS" OR "RBS") AND "X51");
END_REGION

REGION Network 2
   RUNG wire#powerrail
      Contact( "X50" )
      Contact( "X40" )
      Contact( "X70" )
      Contact( "X32" )
      wire#w1
      Coil( "X51" )
   END_RUNG
   RUNG wire#powerrail
      Contact( "X51" )
      I_Contact( "X50" )
   END_RUNG wire#w1
   // the same network as SCL:
   "X51" := ("X50" AND "X40" AND "X70" AND "X32") OR ("X51" AND NOT "X50");
END_REGION
END_FUNCTION

FUNCTION "Auto_SansRB_E" : Void   // FC7, LAD
TITLE = Auto Sans RB Entree
{ S7_Optimized_Access := 'TRUE' }
VERSION : 0.1
   VAR_TEMP   // added for the SCL form of the ladder/FBD networks
      _w1 : Bool;
   END_VAR
BEGIN

REGION Network 1
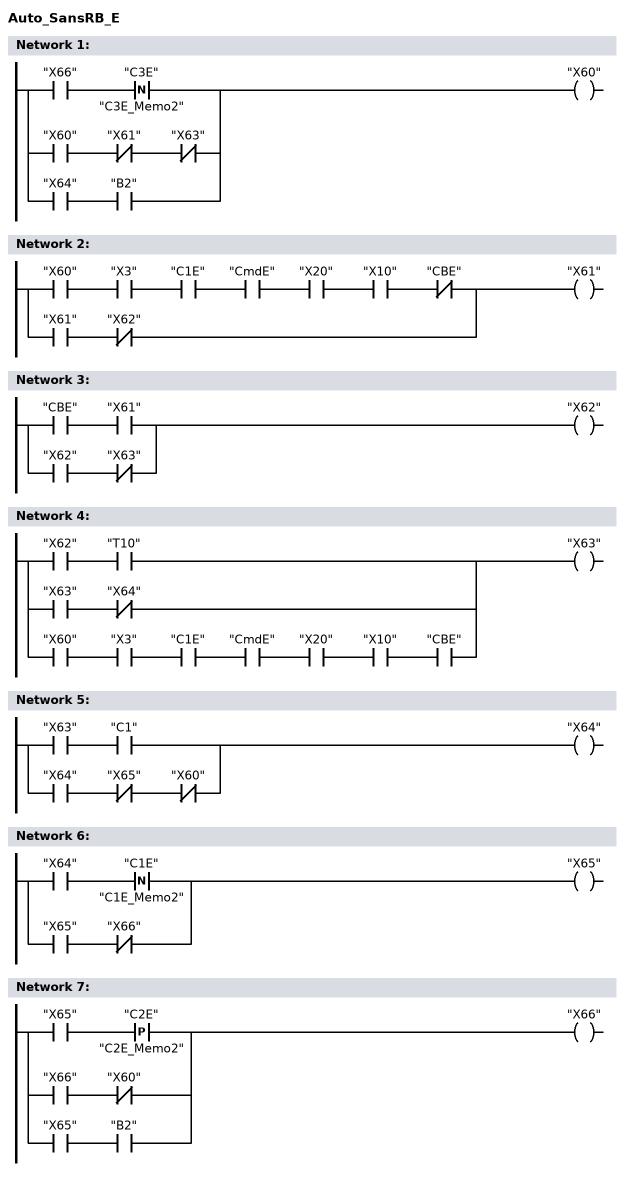
   RUNG wire#powerrail
      Contact( "X66" )
      N_Contact(operand := "C3E", bit := "C3E_Memo2")
      wire#w1
      Coil( "X60" )
   END_RUNG
   RUNG wire#powerrail
      Contact( "X60" )
      I_Contact( "X61" )
      I_Contact( "X63" )
   END_RUNG wire#w1
   RUNG wire#powerrail
      Contact( "X64" )
      Contact( "B2" )
   END_RUNG wire#w1
   // the same network as SCL:
   #_w1 := "X66" AND NOT "C3E" AND "C3E_Memo2";   // falling edge of "C3E"
   "C3E_Memo2" := "C3E";
   "X60" := #_w1 OR ("X60" AND NOT "X61" AND NOT "X63") OR ("X64" AND "B2");
END_REGION

REGION Network 2
   RUNG wire#powerrail
      Contact( "X60" )
      Contact( "X3" )
      Contact( "C1E" )
      Contact( "CmdE" )
      Contact( "X20" )
      Contact( "X10" )
      I_Contact( "CBE" )
      wire#w1
      Coil( "X61" )
   END_RUNG
   RUNG wire#powerrail
      Contact( "X61" )
      I_Contact( "X62" )
   END_RUNG wire#w1
   // the same network as SCL:
   "X61" := ("X60" AND "X3" AND "C1E" AND "CmdE" AND "X20" AND "X10" AND NOT "CBE") OR ("X61" AND NOT "X62");
END_REGION

REGION Network 3
   RUNG wire#powerrail
      Contact( "CBE" )
      Contact( "X61" )
      wire#w1
      Coil( "X62" )
   END_RUNG
   RUNG wire#powerrail
      Contact( "X62" )
      I_Contact( "X63" )
   END_RUNG wire#w1
   // the same network as SCL:
   "X62" := ("CBE" AND "X61") OR ("X62" AND NOT "X63");
END_REGION

REGION Network 4
   RUNG wire#powerrail
      Contact( "X62" )
      Contact( "T10" )
      wire#w1
      Coil( "X63" )
   END_RUNG
   RUNG wire#powerrail
      Contact( "X63" )
      I_Contact( "X64" )
   END_RUNG wire#w1
   RUNG wire#powerrail
      Contact( "X60" )
      Contact( "X3" )
      Contact( "C1E" )
      Contact( "CmdE" )
      Contact( "X20" )
      Contact( "X10" )
      Contact( "CBE" )
   END_RUNG wire#w1
   // the same network as SCL:
   "X63" := ("X62" AND "T10") OR ("X63" AND NOT "X64") OR ("X60" AND "X3" AND "C1E" AND "CmdE" AND "X20" AND "X10" AND "CBE");
END_REGION

REGION Network 5
   RUNG wire#powerrail
      Contact( "X63" )
      Contact( "C1" )
      wire#w1
      Coil( "X64" )
   END_RUNG
   RUNG wire#powerrail
      Contact( "X64" )
      I_Contact( "X65" )
      I_Contact( "X60" )
   END_RUNG wire#w1
   // the same network as SCL:
   "X64" := ("X63" AND "C1") OR ("X64" AND NOT "X65" AND NOT "X60");
END_REGION

REGION Network 6
   RUNG wire#powerrail
      Contact( "X64" )
      N_Contact(operand := "C1E", bit := "C1E_Memo2")
      wire#w1
      Coil( "X65" )
   END_RUNG
   RUNG wire#powerrail
      Contact( "X65" )
      I_Contact( "X66" )
   END_RUNG wire#w1
   // the same network as SCL:
   #_w1 := "X64" AND NOT "C1E" AND "C1E_Memo2";   // falling edge of "C1E"
   "C1E_Memo2" := "C1E";
   "X65" := #_w1 OR ("X65" AND NOT "X66");
END_REGION

REGION Network 7
   RUNG wire#powerrail
      Contact( "X65" )
      P_Contact(operand := "C2E", bit := "C2E_Memo2")
      wire#w1
      Coil( "X66" )
   END_RUNG
   RUNG wire#powerrail
      Contact( "X66" )
      I_Contact( "X60" )
   END_RUNG wire#w1
   RUNG wire#powerrail
      Contact( "X65" )
      Contact( "B2" )
   END_RUNG wire#w1
   // the same network as SCL:
   #_w1 := "X65" AND "C2E" AND NOT "C2E_Memo2";   // rising edge of "C2E"
   "C2E_Memo2" := "C2E";
   "X66" := #_w1 OR ("X66" AND NOT "X60") OR ("X65" AND "B2");
END_REGION
END_FUNCTION

FUNCTION "Auto_SansRB_S" : Void   // FC8, LAD
TITLE = Anto Sans RB Sortie
{ S7_Optimized_Access := 'TRUE' }
VERSION : 0.1
   VAR_TEMP   // added for the SCL form of the ladder/FBD networks
      _w1 : Bool;
   END_VAR
BEGIN

REGION Network 1
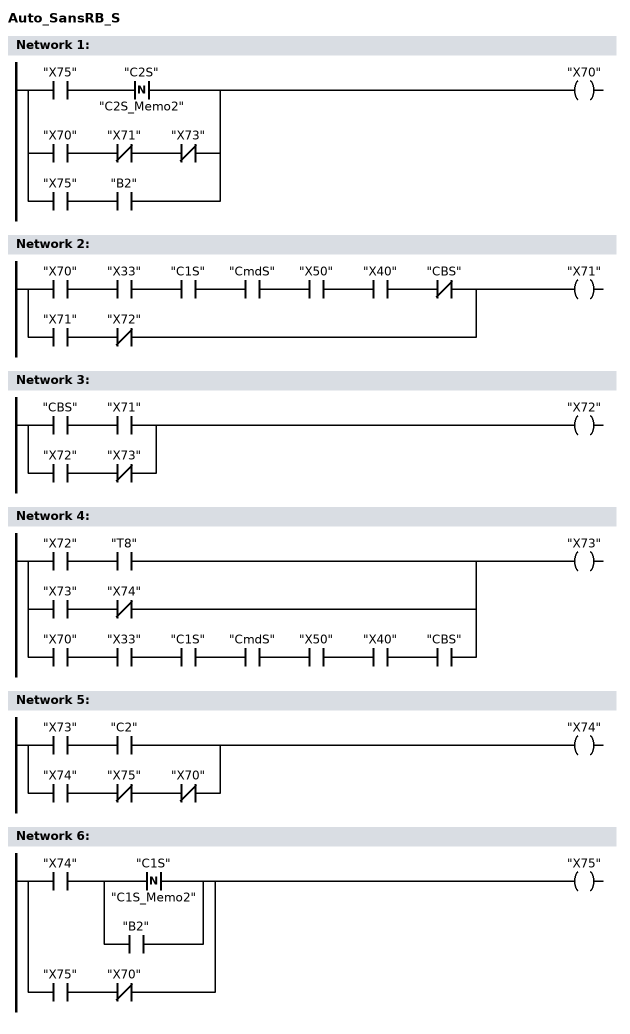
   RUNG wire#powerrail
      Contact( "X75" )
      N_Contact(operand := "C2S", bit := "C2S_Memo2")
      wire#w1
      Coil( "X70" )
   END_RUNG
   RUNG wire#powerrail
      Contact( "X70" )
      I_Contact( "X71" )
      I_Contact( "X73" )
   END_RUNG wire#w1
   RUNG wire#powerrail
      Contact( "X75" )
      Contact( "B2" )
   END_RUNG wire#w1
   // the same network as SCL:
   #_w1 := "X75" AND NOT "C2S" AND "C2S_Memo2";   // falling edge of "C2S"
   "C2S_Memo2" := "C2S";
   "X70" := #_w1 OR ("X70" AND NOT "X71" AND NOT "X73") OR ("X75" AND "B2");
END_REGION

REGION Network 2
   RUNG wire#powerrail
      Contact( "X70" )
      Contact( "X33" )
      Contact( "C1S" )
      Contact( "CmdS" )
      Contact( "X50" )
      Contact( "X40" )
      I_Contact( "CBS" )
      wire#w1
      Coil( "X71" )
   END_RUNG
   RUNG wire#powerrail
      Contact( "X71" )
      I_Contact( "X72" )
   END_RUNG wire#w1
   // the same network as SCL:
   "X71" := ("X70" AND "X33" AND "C1S" AND "CmdS" AND "X50" AND "X40" AND NOT "CBS") OR ("X71" AND NOT "X72");
END_REGION

REGION Network 3
   RUNG wire#powerrail
      Contact( "CBS" )
      Contact( "X71" )
      wire#w1
      Coil( "X72" )
   END_RUNG
   RUNG wire#powerrail
      Contact( "X72" )
      I_Contact( "X73" )
   END_RUNG wire#w1
   // the same network as SCL:
   "X72" := ("CBS" AND "X71") OR ("X72" AND NOT "X73");
END_REGION

REGION Network 4
   RUNG wire#powerrail
      Contact( "X72" )
      Contact( "T8" )
      wire#w1
      Coil( "X73" )
   END_RUNG
   RUNG wire#powerrail
      Contact( "X73" )
      I_Contact( "X74" )
   END_RUNG wire#w1
   RUNG wire#powerrail
      Contact( "X70" )
      Contact( "X33" )
      Contact( "C1S" )
      Contact( "CmdS" )
      Contact( "X50" )
      Contact( "X40" )
      Contact( "CBS" )
   END_RUNG wire#w1
   // the same network as SCL:
   "X73" := ("X72" AND "T8") OR ("X73" AND NOT "X74") OR ("X70" AND "X33" AND "C1S" AND "CmdS" AND "X50" AND "X40" AND "CBS");
END_REGION

REGION Network 5
   RUNG wire#powerrail
      Contact( "X73" )
      Contact( "C2" )
      wire#w1
      Coil( "X74" )
   END_RUNG
   RUNG wire#powerrail
      Contact( "X74" )
      I_Contact( "X75" )
      I_Contact( "X70" )
   END_RUNG wire#w1
   // the same network as SCL:
   "X74" := ("X73" AND "C2") OR ("X74" AND NOT "X75" AND NOT "X70");
END_REGION

REGION Network 6
   RUNG wire#powerrail
      Contact( "X74" )
      wire#w1
      N_Contact(operand := "C1S", bit := "C1S_Memo2")
      wire#w2
      Coil( "X75" )
   END_RUNG
   RUNG wire#w1
      Contact( "B2" )
   END_RUNG wire#w2
   RUNG wire#powerrail
      Contact( "X75" )
      I_Contact( "X70" )
   END_RUNG wire#w2
   // the same network as SCL:
   #_w1 := "X74" AND NOT "C1S" AND "C1S_Memo2";   // falling edge of "C1S"
   "C1S_Memo2" := "C1S";
   "X75" := #_w1 OR ("X74" AND "B2") OR ("X75" AND NOT "X70");
END_REGION
END_FUNCTION

FUNCTION "ImageInput" : Void   // FC9, LAD
{ S7_Optimized_Access := 'TRUE' }
VERSION : 0.1
BEGIN

REGION Network 1: Image entree 0
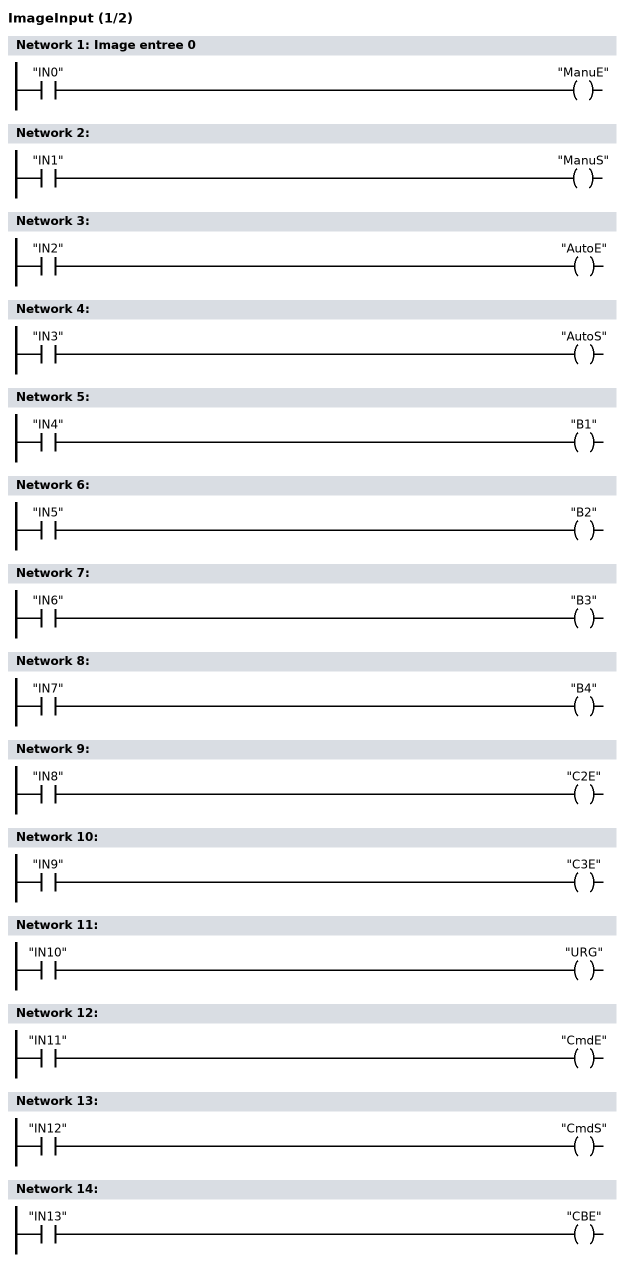
   RUNG wire#powerrail
      Contact( "IN0" )
      Coil( "ManuE" )
   END_RUNG
   // the same network as SCL:
   "ManuE" := "IN0";
END_REGION

REGION Network 2
   RUNG wire#powerrail
      Contact( "IN1" )
      Coil( "ManuS" )
   END_RUNG
   // the same network as SCL:
   "ManuS" := "IN1";
END_REGION

REGION Network 3
   RUNG wire#powerrail
      Contact( "IN2" )
      Coil( "AutoE" )
   END_RUNG
   // the same network as SCL:
   "AutoE" := "IN2";
END_REGION

REGION Network 4
   RUNG wire#powerrail
      Contact( "IN3" )
      Coil( "AutoS" )
   END_RUNG
   // the same network as SCL:
   "AutoS" := "IN3";
END_REGION

REGION Network 5
   RUNG wire#powerrail
      Contact( "IN4" )
      Coil( "B1" )
   END_RUNG
   // the same network as SCL:
   "B1" := "IN4";
END_REGION

REGION Network 6
   RUNG wire#powerrail
      Contact( "IN5" )
      Coil( "B2" )
   END_RUNG
   // the same network as SCL:
   "B2" := "IN5";
END_REGION

REGION Network 7
   RUNG wire#powerrail
      Contact( "IN6" )
      Coil( "B3" )
   END_RUNG
   // the same network as SCL:
   "B3" := "IN6";
END_REGION

REGION Network 8
   RUNG wire#powerrail
      Contact( "IN7" )
      Coil( "B4" )
   END_RUNG
   // the same network as SCL:
   "B4" := "IN7";
END_REGION

REGION Network 9
   RUNG wire#powerrail
      Contact( "IN8" )
      Coil( "C2E" )
   END_RUNG
   // the same network as SCL:
   "C2E" := "IN8";
END_REGION

REGION Network 10
   RUNG wire#powerrail
      Contact( "IN9" )
      Coil( "C3E" )
   END_RUNG
   // the same network as SCL:
   "C3E" := "IN9";
END_REGION

REGION Network 11
   RUNG wire#powerrail
      Contact( "IN10" )
      Coil( "URG" )
   END_RUNG
   // the same network as SCL:
   "URG" := "IN10";
END_REGION

REGION Network 12
   RUNG wire#powerrail
      Contact( "IN11" )
      Coil( "CmdE" )
   END_RUNG
   // the same network as SCL:
   "CmdE" := "IN11";
END_REGION

REGION Network 13
   RUNG wire#powerrail
      Contact( "IN12" )
      Coil( "CmdS" )
   END_RUNG
   // the same network as SCL:
   "CmdS" := "IN12";
END_REGION

REGION Network 14
   RUNG wire#powerrail
      Contact( "IN13" )
      Coil( "CBE" )
   END_RUNG
   // the same network as SCL:
   "CBE" := "IN13";
END_REGION

REGION Network 15
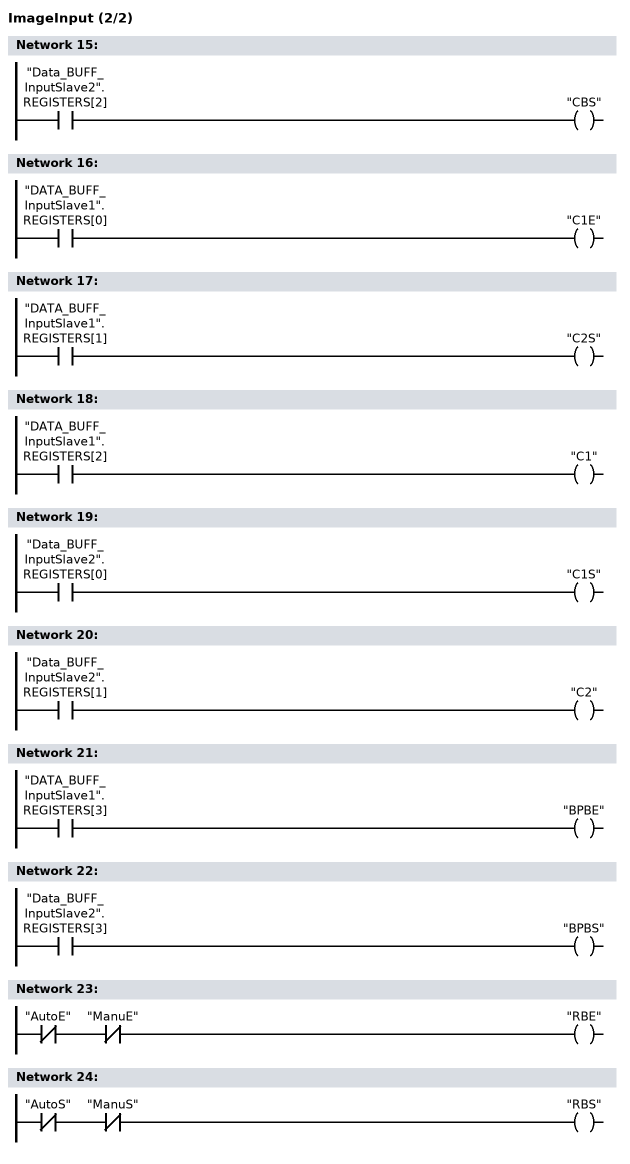
   RUNG wire#powerrail
      Contact( "Data_BUFF_InputSlave2".REGISTERS[2] )
      Coil( "CBS" )
   END_RUNG
   // the same network as SCL:
   "CBS" := "Data_BUFF_InputSlave2".REGISTERS[2];
END_REGION

REGION Network 16
   RUNG wire#powerrail
      Contact( "DATA_BUFF_InputSlave1".REGISTERS[0] )
      Coil( "C1E" )
   END_RUNG
   // the same network as SCL:
   "C1E" := "DATA_BUFF_InputSlave1".REGISTERS[0];
END_REGION

REGION Network 17
   RUNG wire#powerrail
      Contact( "DATA_BUFF_InputSlave1".REGISTERS[1] )
      Coil( "C2S" )
   END_RUNG
   // the same network as SCL:
   "C2S" := "DATA_BUFF_InputSlave1".REGISTERS[1];
END_REGION

REGION Network 18
   RUNG wire#powerrail
      Contact( "DATA_BUFF_InputSlave1".REGISTERS[2] )
      Coil( "C1" )
   END_RUNG
   // the same network as SCL:
   "C1" := "DATA_BUFF_InputSlave1".REGISTERS[2];
END_REGION

REGION Network 19
   RUNG wire#powerrail
      Contact( "Data_BUFF_InputSlave2".REGISTERS[0] )
      Coil( "C1S" )
   END_RUNG
   // the same network as SCL:
   "C1S" := "Data_BUFF_InputSlave2".REGISTERS[0];
END_REGION

REGION Network 20
   RUNG wire#powerrail
      Contact( "Data_BUFF_InputSlave2".REGISTERS[1] )
      Coil( "C2" )
   END_RUNG
   // the same network as SCL:
   "C2" := "Data_BUFF_InputSlave2".REGISTERS[1];
END_REGION

REGION Network 21
   RUNG wire#powerrail
      Contact( "DATA_BUFF_InputSlave1".REGISTERS[3] )
      Coil( "BPBE" )
   END_RUNG
   // the same network as SCL:
   "BPBE" := "DATA_BUFF_InputSlave1".REGISTERS[3];
END_REGION

REGION Network 22
   RUNG wire#powerrail
      Contact( "Data_BUFF_InputSlave2".REGISTERS[3] )
      Coil( "BPBS" )
   END_RUNG
   // the same network as SCL:
   "BPBS" := "Data_BUFF_InputSlave2".REGISTERS[3];
END_REGION

REGION Network 23
   RUNG wire#powerrail
      I_Contact( "AutoE" )
      I_Contact( "ManuE" )
      Coil( "RBE" )
   END_RUNG
   // the same network as SCL:
   "RBE" := NOT "AutoE" AND NOT "ManuE";
END_REGION

REGION Network 24
   RUNG wire#powerrail
      I_Contact( "AutoS" )
      I_Contact( "ManuS" )
      Coil( "RBS" )
   END_RUNG
   // the same network as SCL:
   "RBS" := NOT "AutoS" AND NOT "ManuS";
END_REGION
END_FUNCTION

FUNCTION "ImageOutput" : Void   // FC10, LAD
{ S7_Optimized_Access := 'TRUE' }
VERSION : 0.1
BEGIN

REGION Network 1
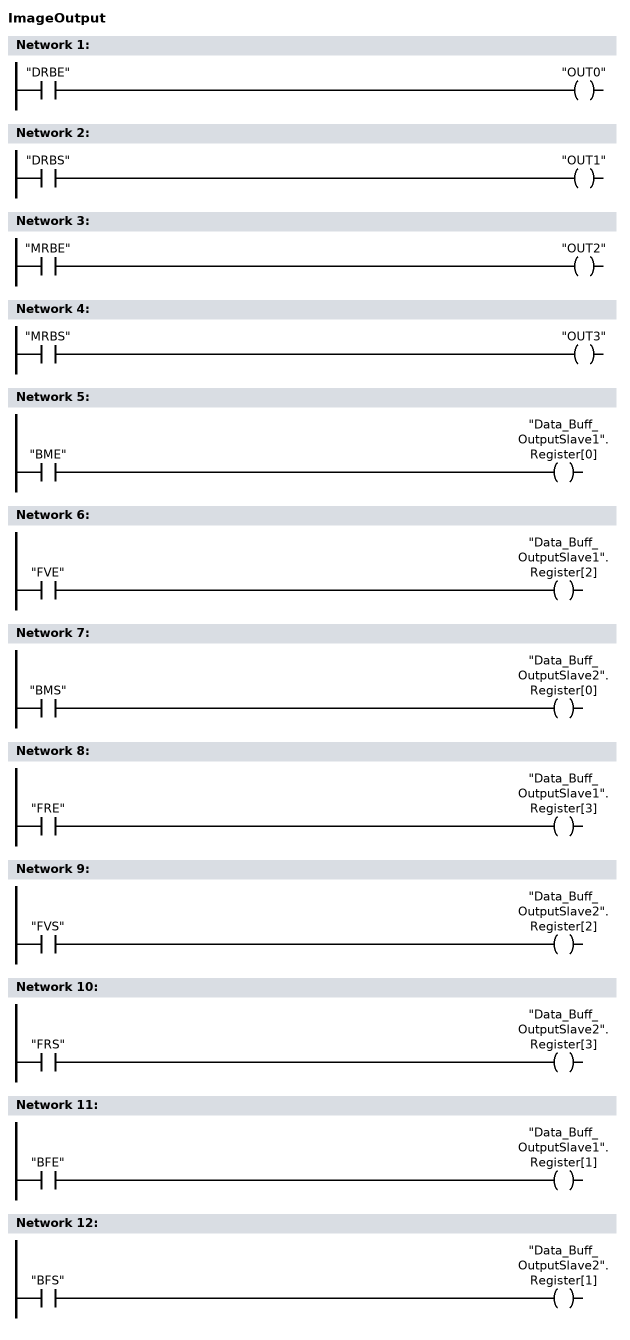
   RUNG wire#powerrail
      Contact( "DRBE" )
      Coil( "OUT0" )
   END_RUNG
   // the same network as SCL:
   "OUT0" := "DRBE";
END_REGION

REGION Network 2
   RUNG wire#powerrail
      Contact( "DRBS" )
      Coil( "OUT1" )
   END_RUNG
   // the same network as SCL:
   "OUT1" := "DRBS";
END_REGION

REGION Network 3
   RUNG wire#powerrail
      Contact( "MRBE" )
      Coil( "OUT2" )
   END_RUNG
   // the same network as SCL:
   "OUT2" := "MRBE";
END_REGION

REGION Network 4
   RUNG wire#powerrail
      Contact( "MRBS" )
      Coil( "OUT3" )
   END_RUNG
   // the same network as SCL:
   "OUT3" := "MRBS";
END_REGION

REGION Network 5
   RUNG wire#powerrail
      Contact( "BME" )
      Coil( "Data_Buff_OutputSlave1".Register[0] )
   END_RUNG
   // the same network as SCL:
   "Data_Buff_OutputSlave1".Register[0] := "BME";
END_REGION

REGION Network 6
   RUNG wire#powerrail
      Contact( "FVE" )
      Coil( "Data_Buff_OutputSlave1".Register[2] )
   END_RUNG
   // the same network as SCL:
   "Data_Buff_OutputSlave1".Register[2] := "FVE";
END_REGION

REGION Network 7
   RUNG wire#powerrail
      Contact( "BMS" )
      Coil( "Data_Buff_OutputSlave2".Register[0] )
   END_RUNG
   // the same network as SCL:
   "Data_Buff_OutputSlave2".Register[0] := "BMS";
END_REGION

REGION Network 8
   RUNG wire#powerrail
      Contact( "FRE" )
      Coil( "Data_Buff_OutputSlave1".Register[3] )
   END_RUNG
   // the same network as SCL:
   "Data_Buff_OutputSlave1".Register[3] := "FRE";
END_REGION

REGION Network 9
   RUNG wire#powerrail
      Contact( "FVS" )
      Coil( "Data_Buff_OutputSlave2".Register[2] )
   END_RUNG
   // the same network as SCL:
   "Data_Buff_OutputSlave2".Register[2] := "FVS";
END_REGION

REGION Network 10
   RUNG wire#powerrail
      Contact( "FRS" )
      Coil( "Data_Buff_OutputSlave2".Register[3] )
   END_RUNG
   // the same network as SCL:
   "Data_Buff_OutputSlave2".Register[3] := "FRS";
END_REGION

REGION Network 11
   RUNG wire#powerrail
      Contact( "BFE" )
      Coil( "Data_Buff_OutputSlave1".Register[1] )
   END_RUNG
   // the same network as SCL:
   "Data_Buff_OutputSlave1".Register[1] := "BFE";
END_REGION

REGION Network 12
   RUNG wire#powerrail
      Contact( "BFS" )
      Coil( "Data_Buff_OutputSlave2".Register[1] )
   END_RUNG
   // the same network as SCL:
   "Data_Buff_OutputSlave2".Register[1] := "BFS";
END_REGION
END_FUNCTION

FUNCTION "AUE" : Void   // FC11, LAD
TITLE = Full Auto Entree
{ S7_Optimized_Access := 'TRUE' }
VERSION : 0.1
   VAR_TEMP   // added for the SCL form of the ladder/FBD networks
      _w1 : Bool;
   END_VAR
BEGIN

REGION Network 1
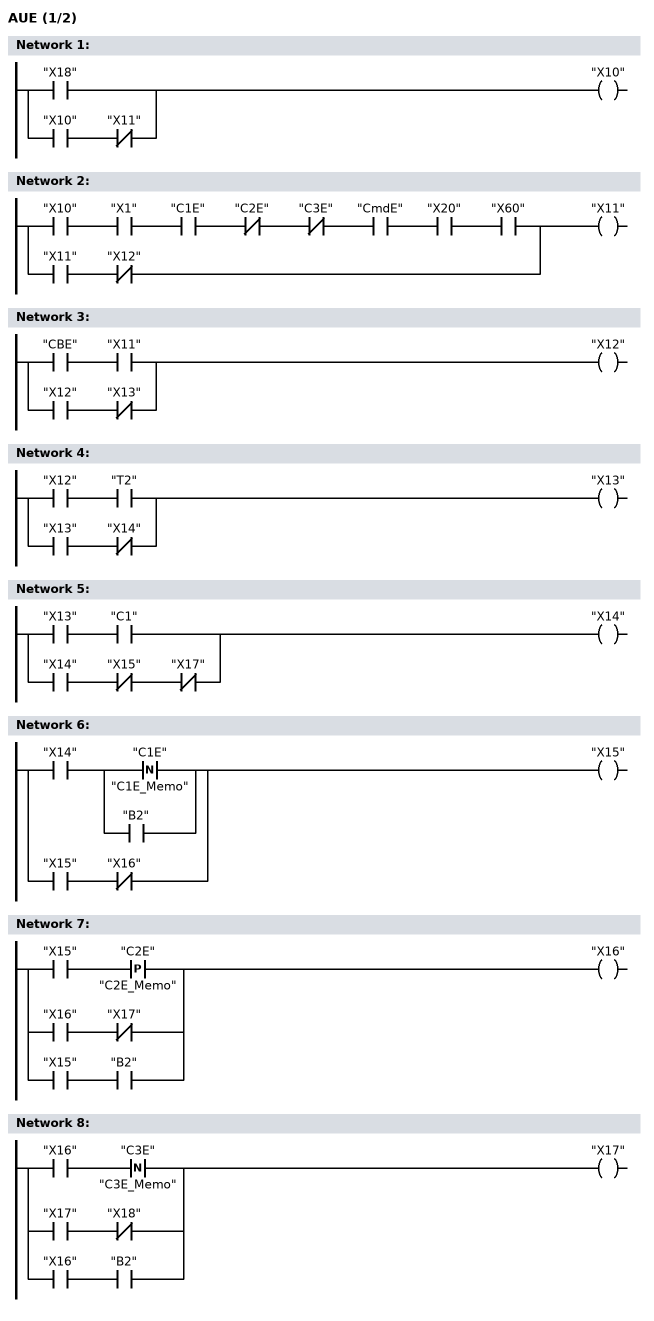
   RUNG wire#powerrail
      Contact( "X18" )
      wire#w1
      Coil( "X10" )
   END_RUNG
   RUNG wire#powerrail
      Contact( "X10" )
      I_Contact( "X11" )
   END_RUNG wire#w1
   // the same network as SCL:
   "X10" := "X18" OR ("X10" AND NOT "X11");
END_REGION

REGION Network 2
   RUNG wire#powerrail
      Contact( "X10" )
      Contact( "X1" )
      Contact( "C1E" )
      I_Contact( "C2E" )
      I_Contact( "C3E" )
      Contact( "CmdE" )
      Contact( "X20" )
      Contact( "X60" )
      wire#w1
      Coil( "X11" )
   END_RUNG
   RUNG wire#powerrail
      Contact( "X11" )
      I_Contact( "X12" )
   END_RUNG wire#w1
   // the same network as SCL:
   "X11" := ("X10" AND "X1" AND "C1E" AND NOT "C2E" AND NOT "C3E" AND "CmdE" AND "X20" AND "X60") OR ("X11" AND NOT "X12");
END_REGION

REGION Network 3
   RUNG wire#powerrail
      Contact( "CBE" )
      Contact( "X11" )
      wire#w1
      Coil( "X12" )
   END_RUNG
   RUNG wire#powerrail
      Contact( "X12" )
      I_Contact( "X13" )
   END_RUNG wire#w1
   // the same network as SCL:
   "X12" := ("CBE" AND "X11") OR ("X12" AND NOT "X13");
END_REGION

REGION Network 4
   RUNG wire#powerrail
      Contact( "X12" )
      Contact( "T2" )
      wire#w1
      Coil( "X13" )
   END_RUNG
   RUNG wire#powerrail
      Contact( "X13" )
      I_Contact( "X14" )
   END_RUNG wire#w1
   // the same network as SCL:
   "X13" := ("X12" AND "T2") OR ("X13" AND NOT "X14");
END_REGION

REGION Network 5
   RUNG wire#powerrail
      Contact( "X13" )
      Contact( "C1" )
      wire#w1
      Coil( "X14" )
   END_RUNG
   RUNG wire#powerrail
      Contact( "X14" )
      I_Contact( "X15" )
      I_Contact( "X17" )
   END_RUNG wire#w1
   // the same network as SCL:
   "X14" := ("X13" AND "C1") OR ("X14" AND NOT "X15" AND NOT "X17");
END_REGION

REGION Network 6
   RUNG wire#powerrail
      Contact( "X14" )
      wire#w1
      N_Contact(operand := "C1E", bit := "C1E_Memo")
      wire#w2
      Coil( "X15" )
   END_RUNG
   RUNG wire#w1
      Contact( "B2" )
   END_RUNG wire#w2
   RUNG wire#powerrail
      Contact( "X15" )
      I_Contact( "X16" )
   END_RUNG wire#w2
   // the same network as SCL:
   #_w1 := "X14" AND NOT "C1E" AND "C1E_Memo";   // falling edge of "C1E"
   "C1E_Memo" := "C1E";
   "X15" := #_w1 OR ("X14" AND "B2") OR ("X15" AND NOT "X16");
END_REGION

REGION Network 7
   RUNG wire#powerrail
      Contact( "X15" )
      P_Contact(operand := "C2E", bit := "C2E_Memo")
      wire#w1
      Coil( "X16" )
   END_RUNG
   RUNG wire#powerrail
      Contact( "X16" )
      I_Contact( "X17" )
   END_RUNG wire#w1
   RUNG wire#powerrail
      Contact( "X15" )
      Contact( "B2" )
   END_RUNG wire#w1
   // the same network as SCL:
   #_w1 := "X15" AND "C2E" AND NOT "C2E_Memo";   // rising edge of "C2E"
   "C2E_Memo" := "C2E";
   "X16" := #_w1 OR ("X16" AND NOT "X17") OR ("X15" AND "B2");
END_REGION

REGION Network 8
   RUNG wire#powerrail
      Contact( "X16" )
      N_Contact(operand := "C3E", bit := "C3E_Memo")
      wire#w1
      Coil( "X17" )
   END_RUNG
   RUNG wire#powerrail
      Contact( "X17" )
      I_Contact( "X18" )
   END_RUNG wire#w1
   RUNG wire#powerrail
      Contact( "X16" )
      Contact( "B2" )
   END_RUNG wire#w1
   // the same network as SCL:
   #_w1 := "X16" AND NOT "C3E" AND "C3E_Memo";   // falling edge of "C3E"
   "C3E_Memo" := "C3E";
   "X17" := #_w1 OR ("X17" AND NOT "X18") OR ("X16" AND "B2");
END_REGION

REGION Network 9
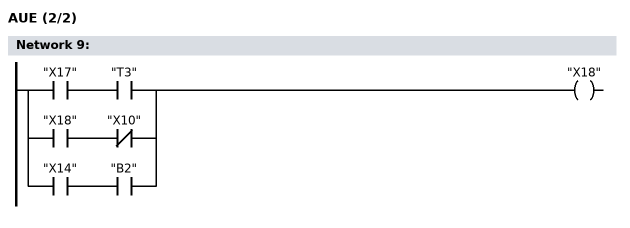
   RUNG wire#powerrail
      Contact( "X17" )
      Contact( "T3" )
      wire#w1
      Coil( "X18" )
   END_RUNG
   RUNG wire#powerrail
      Contact( "X18" )
      I_Contact( "X10" )
   END_RUNG wire#w1
   RUNG wire#powerrail
      Contact( "X14" )
      Contact( "B2" )
   END_RUNG wire#w1
   // the same network as SCL:
   "X18" := ("X17" AND "T3") OR ("X18" AND NOT "X10") OR ("X14" AND "B2");
END_REGION
END_FUNCTION

FUNCTION "AUS" : Void   // FC12, LAD
TITLE = Full Auto Sortie
{ S7_Optimized_Access := 'TRUE' }
VERSION : 0.1
   VAR_TEMP   // added for the SCL form of the ladder/FBD networks
      _w1 : Bool;
   END_VAR
BEGIN

REGION Network 1
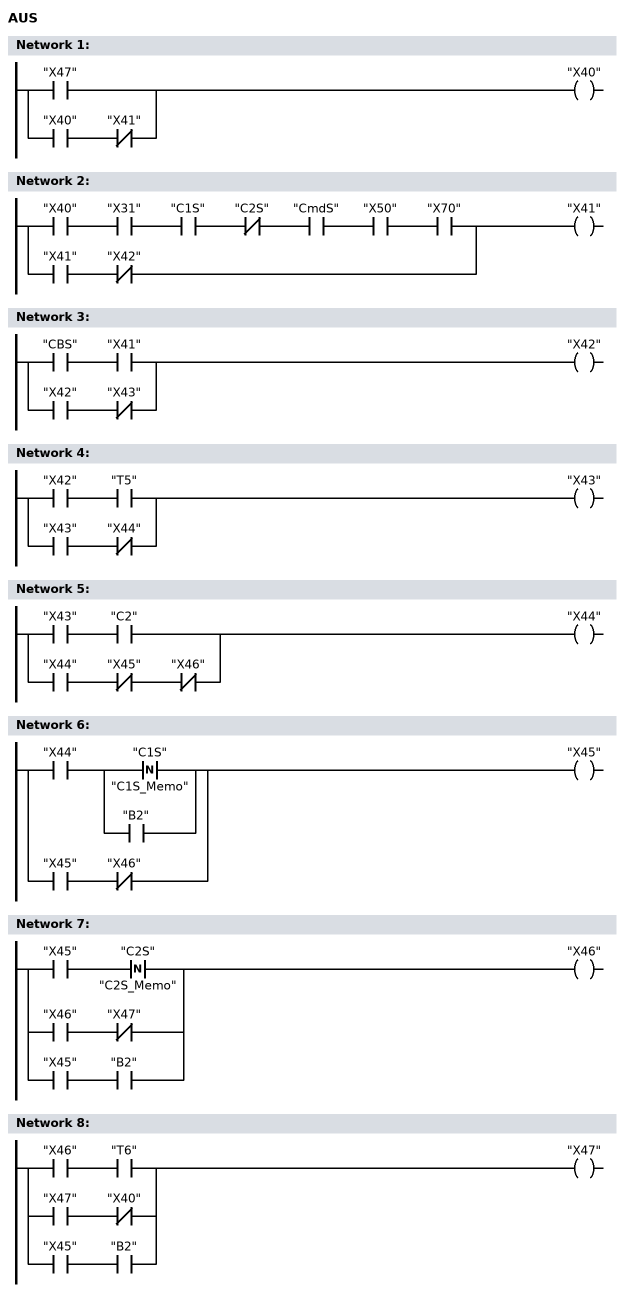
   RUNG wire#powerrail
      Contact( "X47" )
      wire#w1
      Coil( "X40" )
   END_RUNG
   RUNG wire#powerrail
      Contact( "X40" )
      I_Contact( "X41" )
   END_RUNG wire#w1
   // the same network as SCL:
   "X40" := "X47" OR ("X40" AND NOT "X41");
END_REGION

REGION Network 2
   RUNG wire#powerrail
      Contact( "X40" )
      Contact( "X31" )
      Contact( "C1S" )
      I_Contact( "C2S" )
      Contact( "CmdS" )
      Contact( "X50" )
      Contact( "X70" )
      wire#w1
      Coil( "X41" )
   END_RUNG
   RUNG wire#powerrail
      Contact( "X41" )
      I_Contact( "X42" )
   END_RUNG wire#w1
   // the same network as SCL:
   "X41" := ("X40" AND "X31" AND "C1S" AND NOT "C2S" AND "CmdS" AND "X50" AND "X70") OR ("X41" AND NOT "X42");
END_REGION

REGION Network 3
   RUNG wire#powerrail
      Contact( "CBS" )
      Contact( "X41" )
      wire#w1
      Coil( "X42" )
   END_RUNG
   RUNG wire#powerrail
      Contact( "X42" )
      I_Contact( "X43" )
   END_RUNG wire#w1
   // the same network as SCL:
   "X42" := ("CBS" AND "X41") OR ("X42" AND NOT "X43");
END_REGION

REGION Network 4
   RUNG wire#powerrail
      Contact( "X42" )
      Contact( "T5" )
      wire#w1
      Coil( "X43" )
   END_RUNG
   RUNG wire#powerrail
      Contact( "X43" )
      I_Contact( "X44" )
   END_RUNG wire#w1
   // the same network as SCL:
   "X43" := ("X42" AND "T5") OR ("X43" AND NOT "X44");
END_REGION

REGION Network 5
   RUNG wire#powerrail
      Contact( "X43" )
      Contact( "C2" )
      wire#w1
      Coil( "X44" )
   END_RUNG
   RUNG wire#powerrail
      Contact( "X44" )
      I_Contact( "X45" )
      I_Contact( "X46" )
   END_RUNG wire#w1
   // the same network as SCL:
   "X44" := ("X43" AND "C2") OR ("X44" AND NOT "X45" AND NOT "X46");
END_REGION

REGION Network 6
   RUNG wire#powerrail
      Contact( "X44" )
      wire#w1
      N_Contact(operand := "C1S", bit := "C1S_Memo")
      wire#w2
      Coil( "X45" )
   END_RUNG
   RUNG wire#w1
      Contact( "B2" )
   END_RUNG wire#w2
   RUNG wire#powerrail
      Contact( "X45" )
      I_Contact( "X46" )
   END_RUNG wire#w2
   // the same network as SCL:
   #_w1 := "X44" AND NOT "C1S" AND "C1S_Memo";   // falling edge of "C1S"
   "C1S_Memo" := "C1S";
   "X45" := #_w1 OR ("X44" AND "B2") OR ("X45" AND NOT "X46");
END_REGION

REGION Network 7
   RUNG wire#powerrail
      Contact( "X45" )
      N_Contact(operand := "C2S", bit := "C2S_Memo")
      wire#w1
      Coil( "X46" )
   END_RUNG
   RUNG wire#powerrail
      Contact( "X46" )
      I_Contact( "X47" )
   END_RUNG wire#w1
   RUNG wire#powerrail
      Contact( "X45" )
      Contact( "B2" )
   END_RUNG wire#w1
   // the same network as SCL:
   #_w1 := "X45" AND NOT "C2S" AND "C2S_Memo";   // falling edge of "C2S"
   "C2S_Memo" := "C2S";
   "X46" := #_w1 OR ("X46" AND NOT "X47") OR ("X45" AND "B2");
END_REGION

REGION Network 8
   RUNG wire#powerrail
      Contact( "X46" )
      Contact( "T6" )
      wire#w1
      Coil( "X47" )
   END_RUNG
   RUNG wire#powerrail
      Contact( "X47" )
      I_Contact( "X40" )
   END_RUNG wire#w1
   RUNG wire#powerrail
      Contact( "X45" )
      Contact( "B2" )
   END_RUNG wire#w1
   // the same network as SCL:
   "X47" := ("X46" AND "T6") OR ("X47" AND NOT "X40") OR ("X45" AND "B2");
END_REGION
END_FUNCTION

FUNCTION "URGENCE" : Void   // FC13, LAD
{ S7_Optimized_Access := 'TRUE' }
VERSION : 0.1
BEGIN

REGION Network 1
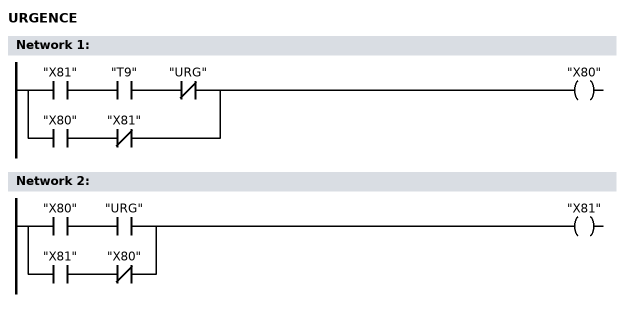
   RUNG wire#powerrail
      Contact( "X81" )
      Contact( "T9" )
      I_Contact( "URG" )
      wire#w1
      Coil( "X80" )
   END_RUNG
   RUNG wire#powerrail
      Contact( "X80" )
      I_Contact( "X81" )
   END_RUNG wire#w1
   // the same network as SCL:
   "X80" := ("X81" AND "T9" AND NOT "URG") OR ("X80" AND NOT "X81");
END_REGION

REGION Network 2
   RUNG wire#powerrail
      Contact( "X80" )
      Contact( "URG" )
      wire#w1
      Coil( "X81" )
   END_RUNG
   RUNG wire#powerrail
      Contact( "X81" )
      I_Contact( "X80" )
   END_RUNG wire#w1
   // the same network as SCL:
   "X81" := ("X80" AND "URG") OR ("X81" AND NOT "X80");
END_REGION
END_FUNCTION

FUNCTION "Actions" : Void   // FC14, LAD
{ S7_Optimized_Access := 'TRUE' }
VERSION : 0.1
   VAR_TEMP   // added for the SCL form of the ladder/FBD networks
      _w1 : Bool;
      _w2 : Bool;
   END_VAR
BEGIN

REGION Network 1
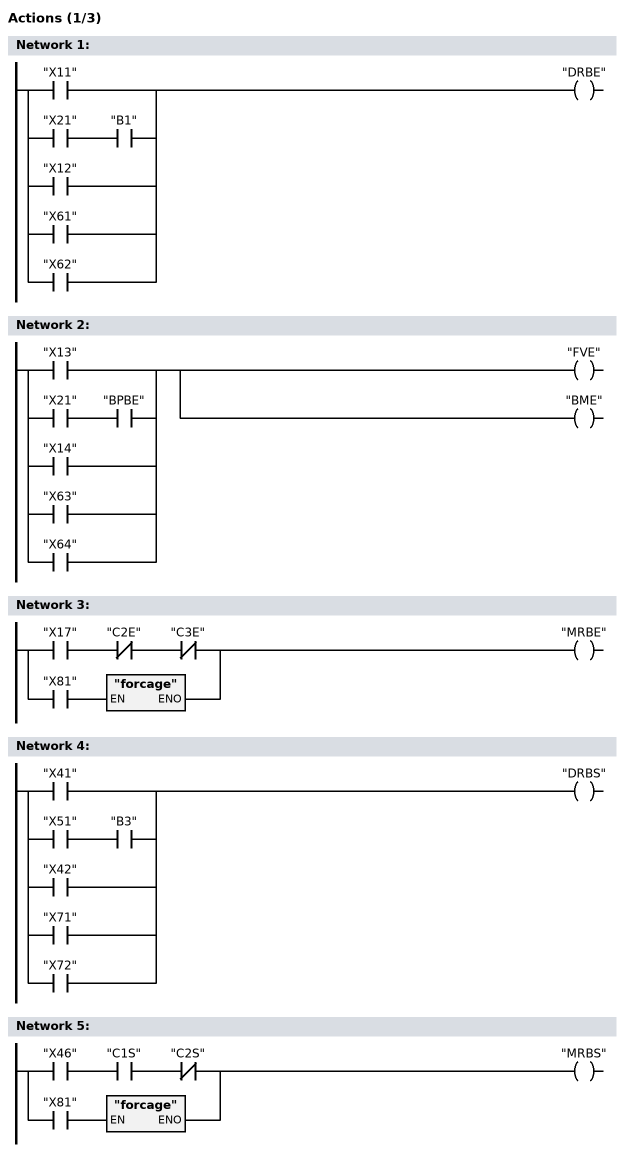
   RUNG wire#powerrail
      Contact( "X11" )
      wire#w1
      Coil( "DRBE" )
   END_RUNG
   RUNG wire#powerrail
      Contact( "X21" )
      Contact( "B1" )
   END_RUNG wire#w1
   RUNG wire#powerrail
      Contact( "X12" )
   END_RUNG wire#w1
   RUNG wire#powerrail
      Contact( "X61" )
   END_RUNG wire#w1
   RUNG wire#powerrail
      Contact( "X62" )
   END_RUNG wire#w1
   // the same network as SCL:
   "DRBE" := "X11" OR ("X21" AND "B1") OR "X12" OR "X61" OR "X62";
END_REGION

REGION Network 2
   RUNG wire#powerrail
      Contact( "X13" )
      wire#w1
      Coil( "FVE" )
   END_RUNG
   RUNG wire#powerrail
      Contact( "X21" )
      Contact( "BPBE" )
   END_RUNG wire#w1
   RUNG wire#powerrail
      Contact( "X14" )
   END_RUNG wire#w1
   RUNG wire#powerrail
      Contact( "X63" )
   END_RUNG wire#w1
   RUNG wire#powerrail
      Contact( "X64" )
   END_RUNG wire#w1
   RUNG wire#w1
      Coil( "BME" )
   END_RUNG
   // the same network as SCL:
   "FVE" := "X13" OR ("X21" AND "BPBE") OR "X14" OR "X63" OR "X64";
   "BME" := "FVE";
END_REGION

REGION Network 3
   RUNG wire#powerrail
      Contact( "X17" )
      I_Contact( "C2E" )
      I_Contact( "C3E" )
      wire#w1
      Coil( "MRBE" )
   END_RUNG
   RUNG wire#powerrail
      Contact( "X81" )
      "forcage"()
   END_RUNG wire#w1
   // the same network as SCL:
   #_w2 := "X17" AND NOT "C2E" AND NOT "C3E";
   "forcage"(EN := "X81", ENO => #_w1);
   "MRBE" := #_w2 OR #_w1;
END_REGION

REGION Network 4
   RUNG wire#powerrail
      Contact( "X41" )
      wire#w1
      Coil( "DRBS" )
   END_RUNG
   RUNG wire#powerrail
      Contact( "X51" )
      Contact( "B3" )
   END_RUNG wire#w1
   RUNG wire#powerrail
      Contact( "X42" )
   END_RUNG wire#w1
   RUNG wire#powerrail
      Contact( "X71" )
   END_RUNG wire#w1
   RUNG wire#powerrail
      Contact( "X72" )
   END_RUNG wire#w1
   // the same network as SCL:
   "DRBS" := "X41" OR ("X51" AND "B3") OR "X42" OR "X71" OR "X72";
END_REGION

REGION Network 5
   RUNG wire#powerrail
      Contact( "X46" )
      Contact( "C1S" )
      I_Contact( "C2S" )
      wire#w1
      Coil( "MRBS" )
   END_RUNG
   RUNG wire#powerrail
      Contact( "X81" )
      "forcage"()
   END_RUNG wire#w1
   // the same network as SCL:
   #_w2 := "X46" AND "C1S" AND NOT "C2S";
   "forcage"(EN := "X81", ENO => #_w1);
   "MRBS" := #_w2 OR #_w1;
END_REGION

REGION Network 6
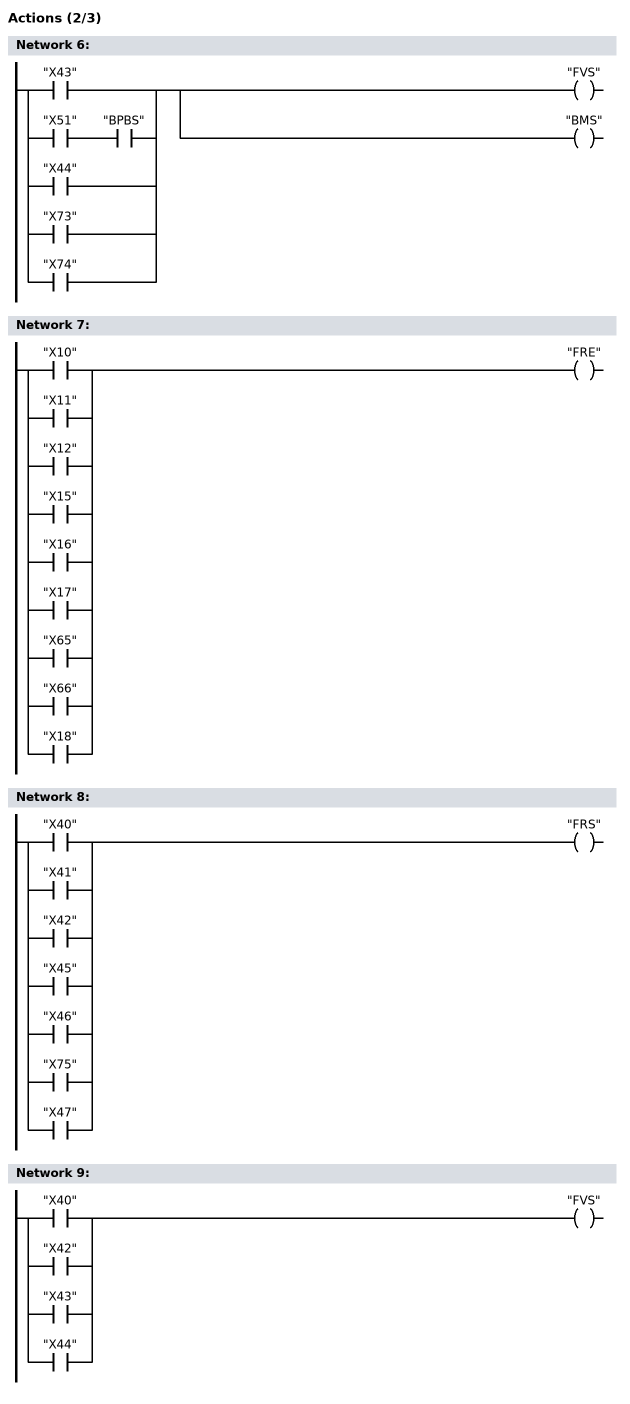
   RUNG wire#powerrail
      Contact( "X43" )
      wire#w1
      Coil( "FVS" )
   END_RUNG
   RUNG wire#powerrail
      Contact( "X51" )
      Contact( "BPBS" )
   END_RUNG wire#w1
   RUNG wire#powerrail
      Contact( "X44" )
   END_RUNG wire#w1
   RUNG wire#powerrail
      Contact( "X73" )
   END_RUNG wire#w1
   RUNG wire#powerrail
      Contact( "X74" )
   END_RUNG wire#w1
   RUNG wire#w1
      Coil( "BMS" )
   END_RUNG
   // the same network as SCL:
   "FVS" := "X43" OR ("X51" AND "BPBS") OR "X44" OR "X73" OR "X74";
   "BMS" := "FVS";
END_REGION

REGION Network 7
   RUNG wire#powerrail
      Contact( "X10" )
      wire#w1
      Coil( "FRE" )
   END_RUNG
   RUNG wire#powerrail
      Contact( "X11" )
   END_RUNG wire#w1
   RUNG wire#powerrail
      Contact( "X12" )
   END_RUNG wire#w1
   RUNG wire#powerrail
      Contact( "X15" )
   END_RUNG wire#w1
   RUNG wire#powerrail
      Contact( "X16" )
   END_RUNG wire#w1
   RUNG wire#powerrail
      Contact( "X17" )
   END_RUNG wire#w1
   RUNG wire#powerrail
      Contact( "X65" )
   END_RUNG wire#w1
   RUNG wire#powerrail
      Contact( "X66" )
   END_RUNG wire#w1
   RUNG wire#powerrail
      Contact( "X18" )
   END_RUNG wire#w1
   // the same network as SCL:
   "FRE" := "X10" OR "X11" OR "X12" OR "X15" OR "X16" OR "X17" OR "X65" OR "X66" OR "X18";
END_REGION

REGION Network 8
   RUNG wire#powerrail
      Contact( "X40" )
      wire#w1
      Coil( "FRS" )
   END_RUNG
   RUNG wire#powerrail
      Contact( "X41" )
   END_RUNG wire#w1
   RUNG wire#powerrail
      Contact( "X42" )
   END_RUNG wire#w1
   RUNG wire#powerrail
      Contact( "X45" )
   END_RUNG wire#w1
   RUNG wire#powerrail
      Contact( "X46" )
   END_RUNG wire#w1
   RUNG wire#powerrail
      Contact( "X75" )
   END_RUNG wire#w1
   RUNG wire#powerrail
      Contact( "X47" )
   END_RUNG wire#w1
   // the same network as SCL:
   "FRS" := "X40" OR "X41" OR "X42" OR "X45" OR "X46" OR "X75" OR "X47";
END_REGION

REGION Network 9
   RUNG wire#powerrail
      Contact( "X40" )
      wire#w1
      Coil( "FVS" )
   END_RUNG
   RUNG wire#powerrail
      Contact( "X42" )
   END_RUNG wire#w1
   RUNG wire#powerrail
      Contact( "X43" )
   END_RUNG wire#w1
   RUNG wire#powerrail
      Contact( "X44" )
   END_RUNG wire#w1
   // the same network as SCL:
   "FVS" := "X40" OR "X42" OR "X43" OR "X44";
END_REGION

REGION Network 10
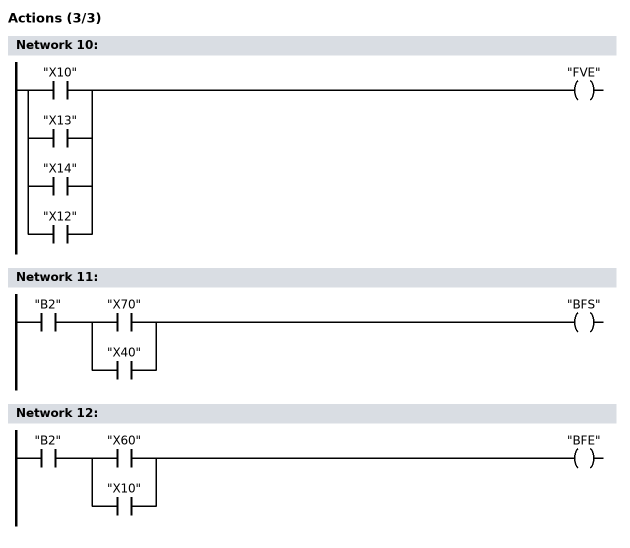
   RUNG wire#powerrail
      Contact( "X10" )
      wire#w1
      Coil( "FVE" )
   END_RUNG
   RUNG wire#powerrail
      Contact( "X13" )
   END_RUNG wire#w1
   RUNG wire#powerrail
      Contact( "X14" )
   END_RUNG wire#w1
   RUNG wire#powerrail
      Contact( "X12" )
   END_RUNG wire#w1
   // the same network as SCL:
   "FVE" := "X10" OR "X13" OR "X14" OR "X12";
END_REGION

REGION Network 11
   RUNG wire#powerrail
      Contact( "B2" )
      wire#w1
      Contact( "X70" )
      wire#w2
      Coil( "BFS" )
   END_RUNG
   RUNG wire#w1
      Contact( "X40" )
   END_RUNG wire#w2
   // the same network as SCL:
   "BFS" := "B2" AND ("X70" OR "X40");
END_REGION

REGION Network 12
   RUNG wire#powerrail
      Contact( "B2" )
      wire#w1
      Contact( "X60" )
      wire#w2
      Coil( "BFE" )
   END_RUNG
   RUNG wire#w1
      Contact( "X10" )
   END_RUNG wire#w2
   // the same network as SCL:
   "BFE" := "B2" AND ("X60" OR "X10");
END_REGION
END_FUNCTION

FUNCTION "forcage" : Void   // FC15, LAD
{ S7_Optimized_Access := 'TRUE' }
VERSION : 0.1
BEGIN

REGION Network 1
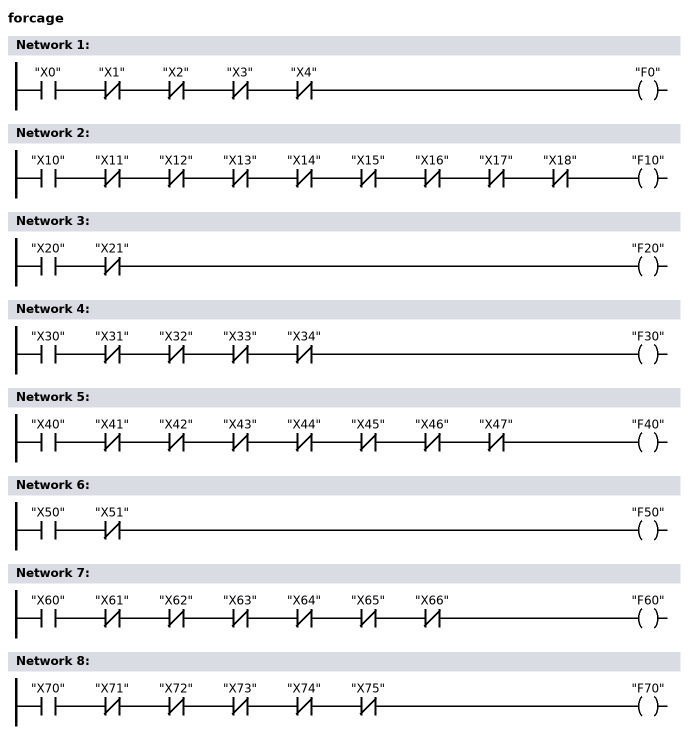
   RUNG wire#powerrail
      Contact( "X0" )
      I_Contact( "X1" )
      I_Contact( "X2" )
      I_Contact( "X3" )
      I_Contact( "X4" )
      Coil( "F0" )
   END_RUNG
   // the same network as SCL:
   "F0" := "X0" AND NOT "X1" AND NOT "X2" AND NOT "X3" AND NOT "X4";
END_REGION

REGION Network 2
   RUNG wire#powerrail
      Contact( "X10" )
      I_Contact( "X11" )
      I_Contact( "X12" )
      I_Contact( "X13" )
      I_Contact( "X14" )
      I_Contact( "X15" )
      I_Contact( "X16" )
      I_Contact( "X17" )
      I_Contact( "X18" )
      Coil( "F10" )
   END_RUNG
   // the same network as SCL:
   "F10" := "X10" AND NOT "X11" AND NOT "X12" AND NOT "X13" AND NOT "X14" AND NOT "X15" AND NOT "X16" AND NOT "X17" AND NOT "X18";
END_REGION

REGION Network 3
   RUNG wire#powerrail
      Contact( "X20" )
      I_Contact( "X21" )
      Coil( "F20" )
   END_RUNG
   // the same network as SCL:
   "F20" := "X20" AND NOT "X21";
END_REGION

REGION Network 4
   RUNG wire#powerrail
      Contact( "X30" )
      I_Contact( "X31" )
      I_Contact( "X32" )
      I_Contact( "X33" )
      I_Contact( "X34" )
      Coil( "F30" )
   END_RUNG
   // the same network as SCL:
   "F30" := "X30" AND NOT "X31" AND NOT "X32" AND NOT "X33" AND NOT "X34";
END_REGION

REGION Network 5
   RUNG wire#powerrail
      Contact( "X40" )
      I_Contact( "X41" )
      I_Contact( "X42" )
      I_Contact( "X43" )
      I_Contact( "X44" )
      I_Contact( "X45" )
      I_Contact( "X46" )
      I_Contact( "X47" )
      Coil( "F40" )
   END_RUNG
   // the same network as SCL:
   "F40" := "X40" AND NOT "X41" AND NOT "X42" AND NOT "X43" AND NOT "X44" AND NOT "X45" AND NOT "X46" AND NOT "X47";
END_REGION

REGION Network 6
   RUNG wire#powerrail
      Contact( "X50" )
      I_Contact( "X51" )
      Coil( "F50" )
   END_RUNG
   // the same network as SCL:
   "F50" := "X50" AND NOT "X51";
END_REGION

REGION Network 7
   RUNG wire#powerrail
      Contact( "X60" )
      I_Contact( "X61" )
      I_Contact( "X62" )
      I_Contact( "X63" )
      I_Contact( "X64" )
      I_Contact( "X65" )
      I_Contact( "X66" )
      Coil( "F60" )
   END_RUNG
   // the same network as SCL:
   "F60" := "X60" AND NOT "X61" AND NOT "X62" AND NOT "X63" AND NOT "X64" AND NOT "X65" AND NOT "X66";
END_REGION

REGION Network 8
   RUNG wire#powerrail
      Contact( "X70" )
      I_Contact( "X71" )
      I_Contact( "X72" )
      I_Contact( "X73" )
      I_Contact( "X74" )
      I_Contact( "X75" )
      Coil( "F70" )
   END_RUNG
   // the same network as SCL:
   "F70" := "X70" AND NOT "X71" AND NOT "X72" AND NOT "X73" AND NOT "X74" AND NOT "X75";
END_REGION
END_FUNCTION

FUNCTION "Temporisation" : Void   // FC16, LAD
{ S7_Optimized_Access := 'TRUE' }
VERSION : 0.1
BEGIN

REGION Network 1
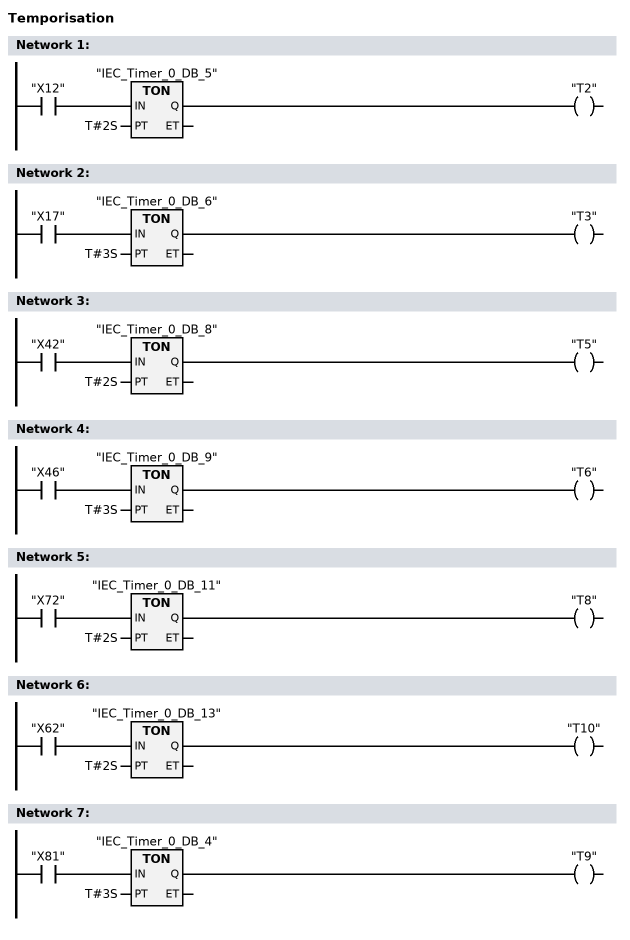
   "IEC_Timer_0_DB_5".TON(IN := "X12", PT := T#2S);
   "T2" := "IEC_Timer_0_DB_5".Q;
END_REGION

REGION Network 2
   "IEC_Timer_0_DB_6".TON(IN := "X17", PT := T#3S);
   "T3" := "IEC_Timer_0_DB_6".Q;
END_REGION

REGION Network 3
   "IEC_Timer_0_DB_8".TON(IN := "X42", PT := T#2S);
   "T5" := "IEC_Timer_0_DB_8".Q;
END_REGION

REGION Network 4
   "IEC_Timer_0_DB_9".TON(IN := "X46", PT := T#3S);
   "T6" := "IEC_Timer_0_DB_9".Q;
END_REGION

REGION Network 5
   "IEC_Timer_0_DB_11".TON(IN := "X72", PT := T#2S);
   "T8" := "IEC_Timer_0_DB_11".Q;
END_REGION

REGION Network 6
   "IEC_Timer_0_DB_13".TON(IN := "X62", PT := T#2S);
   "T10" := "IEC_Timer_0_DB_13".Q;
END_REGION

REGION Network 7
   "IEC_Timer_0_DB_4".TON(IN := "X81", PT := T#3S);
   "T9" := "IEC_Timer_0_DB_4".Q;
END_REGION
END_FUNCTION

FUNCTION "gestion CMD" : Void   // FC17, LAD
{ S7_Optimized_Access := 'TRUE' }
VERSION : 0.1
   VAR_TEMP   // added for the SCL form of the ladder/FBD networks
      _w1 : Bool;
      _w2 : Bool;
   END_VAR
BEGIN

REGION Network 1
